LIN {X 91.990,Y -27.379,Z -185.770,A -90.000,B 90.000,C 0.000} C_DIS
LIN {X 91.908,Y -27.404,Z -186.279,A -90.000,B 90.000,C 0.000} C_DIS
LIN {X 91.890,Y -27.409,Z -186.423,A -90.000,B 90.000,C 0.000} C_DIS
LIN {X 91.690,Y -27.464,Z -187.831,A -90.000,B 90.000,C 0.000} C_DIS
LIN {X 91.648,Y -27.479,Z -188.136,A -90.000,B 90.000,C 0.000} C_DIS
LIN {X 91.626,Y -27.484,Z -188.383,A -90.000,B 90.000,C 0.000} C_DIS
LIN {X 91.538,Y -27.498,Z -189.497,A -90.000,B 90.000,C 0.000} C_DIS
LIN {X 91.494,Y -27.511,Z -190.085,A -90.000,B 90.000,C 0.000} C_DIS
LIN {X 91.464,Y -27.521,Z -190.421,A -90.000,B 90.000,C 0.000} C_DIS
LIN {X 91.445,Y -27.529,Z -190.604,A -90.000,B 90.000,C 0.000} C_DIS
LIN {X 91.394,Y -27.540,Z -191.043,A -90.000,B 90.000,C 0.000} C_DIS
LIN {X 91.332,Y -27.547,Z -191.830,A -90.000,B 90.000,C 0.000} C_DIS
LIN {X 91.227,Y -27.567,Z -193.196,A -90.000,B 90.000,C 0.000} C_DIS
LIN {X 91.184,Y -27.565,Z -193.656,A -90.000,B 90.000,C 0.000} C_DIS
LIN {X 90.969,Y -27.575,Z -195.817,A -90.000,B 90.000,C 0.000} C_DIS
LIN {X 90.925,Y -27.569,Z -196.389,A -90.000,B 90.000,C 0.000} C_DIS
LIN {X 90.877,Y -27.563,Z -196.833,A -90.000,B 90.000,C 0.000} C_DIS
LIN {X 90.590,Y -27.556,Z -198.905,A -90.000,B 90.000,C 0.000} C_DIS
LIN {X 90.465,Y -27.542,Z -199.948,A -90.000,B 90.000,C 0.000} C_DIS
LIN {X 90.447,Y -27.538,Z -200.085,A -90.000,B 90.000,C 0.000} C_DIS
LIN {X 90.408,Y -27.527,Z -200.354,A -90.000,B 90.000,C 0.000} C_DIS
LIN {X 90.390,Y -27.524,Z -200.463,A -90.000,B 90.000,C 0.000} C_DIS
LIN {X 90.100,Y -27.495,Z -202.020,A -90.000,B 90.000,C 0.000} C_DIS
LIN {X 89.684,Y -27.430,Z -204.401,A -90.000,B 90.000,C 0.000} C_DIS
LIN {X 89.653,Y -27.425,Z -204.568,A -90.000,B 90.000,C 0.000} C_DIS
LIN {X 89.484,Y -27.409,Z -205.376,A -90.000,B 90.000,C 0.000} C_DIS
LIN {X 88.923,Y -27.339,Z -208.174,A -90.000,B 90.000,C 0.000} C_DIS
LIN {X 88.721,Y -27.328,Z -209.087,A -90.000,B 90.000,C 0.000} C_DIS
LIN {X 88.664,Y -27.324,Z -209.342,A -90.000,B 90.000,C 0.000} C_DIS
LIN {X 88.255,Y -27.308,Z -211.076,A -90.000,B 90.000,C 0.000} C_DIS
LIN {X 88.255,Y -60.000,Z -211.076,A -90.000,B 90.000,C 0.000} C_DIS
LIN {X -103.369,Y -60.000,Z -243.561,A -90.000,B 90.000,C 0.000} C_DIS
LIN {X -103.369,Y -27.806,Z -243.561,A -90.000,B 90.000,C 0.000} C_DIS
LIN {X -103.055,Y -27.609,Z -243.240,A -90.000,B 90.000,C 0.000} C_DIS
LIN {X -102.608,Y -27.516,Z -242.873,A -90.000,B 90.000,C 0.000} C_DIS
LIN {X -101.362,Y -27.506,Z -241.971,A -90.000,B 90.000,C 0.000} C_DIS
LIN {X -101.122,Y -27.501,Z -241.807,A -90.000,B 90.000,C 0.000} C_DIS
LIN {X -99.449,Y -27.495,Z -240.683,A -90.000,B 90.000,C 0.000} C_DIS
LIN {X -96.335,Y -27.500,Z -238.546,A -90.000,B 90.000,C 0.000} C_DIS
LIN {X -93.712,Y -27.488,Z -236.739,A -90.000,B 90.000,C 0.000} C_DIS
LIN {X -93.290,Y -27.484,Z -236.461,A -90.000,B 90.000,C 0.000} C_DIS
LIN {X -92.213,Y -27.482,Z -235.765,A -90.000,B 90.000,C 0.000} C_DIS
LIN {X -90.517,Y -27.487,Z -234.652,A -90.000,B 90.000,C 0.000} C_DIS
LIN {X -85.124,Y -27.476,Z -231.104,A -90.000,B 90.000,C 0.000} C_DIS
LIN {X -84.873,Y -27.473,Z -230.946,A -90.000,B 90.000,C 0.000} C_DIS
LIN {X -84.774,Y -27.475,Z -230.885,A -90.000,B 90.000,C 0.000} C_DIS
LIN {X -84.558,Y -27.474,Z -230.749,A -90.000,B 90.000,C 0.000} C_DIS
LIN {X -82.273,Y -27.472,Z -229.327,A -90.000,B 90.000,C 0.000} C_DIS
LIN {X -78.940,Y -27.469,Z -227.252,A -90.000,B 90.000,C 0.000} C_DIS
LIN {X -76.872,Y -27.469,Z -225.965,A -90.000,B 90.000,C 0.000} C_DIS
LIN {X -76.380,Y -27.464,Z -225.673,A -90.000,B 90.000,C 0.000} C_DIS
LIN {X -70.507,Y -27.476,Z -222.219,A -90.000,B 90.000,C 0.000} C_DIS
LIN {X -68.311,Y -27.485,Z -220.933,A -90.000,B 90.000,C 0.000} C_DIS
LIN {X -67.723,Y -27.484,Z -220.599,A -90.000,B 90.000,C 0.000} C_DIS
LIN {X -61.693,Y -27.522,Z -217.200,A -90.000,B 90.000,C 0.000} C_DIS
LIN {X -59.270,Y -27.530,Z -215.854,A -90.000,B 90.000,C 0.000} C_DIS
LIN {X -55.292,Y -27.561,Z -213.671,A -90.000,B 90.000,C 0.000} C_DIS
LIN {X -53.229,Y -27.571,Z -212.555,A -90.000,B 90.000,C 0.000} C_DIS
LIN {X -51.847,Y -27.581,Z -211.815,A -90.000,B 90.000,C 0.000} C_DIS
LIN {X -47.655,Y -27.617,Z -209.542,A -90.000,B 90.000,C 0.000} C_DIS
LIN {X -44.795,Y -27.636,Z -208.026,A -90.000,B 90.000,C 0.000} C_DIS
LIN {X -44.368,Y -27.643,Z -207.794,A -90.000,B 90.000,C 0.000} C_DIS
LIN {X -42.572,Y -27.654,Z -206.808,A -90.000,B 90.000,C 0.000} C_DIS
LIN {X -38.988,Y -27.667,Z -204.858,A -90.000,B 90.000,C 0.000} C_DIS
LIN {X -38.628,Y -27.672,Z -204.656,A -90.000,B 90.000,C 0.000} C_DIS
LIN {X -38.069,Y -27.674,Z -204.339,A -90.000,B 90.000,C 0.000} C_DIS
LIN {X -34.183,Y -27.676,Z -202.130,A -90.000,B 90.000,C 0.000} C_DIS
LIN {X -33.519,Y -27.677,Z -201.729,A -90.000,B 90.000,C 0.000} C_DIS
LIN {X -30.256,Y -27.674,Z -199.760,A -90.000,B 90.000,C 0.000} C_DIS
LIN {X -30.194,Y -27.675,Z -199.720,A -90.000,B 90.000,C 0.000} C_DIS
LIN {X -26.908,Y -27.672,Z -197.578,A -90.000,B 90.000,C 0.000} C_DIS
LIN {X -26.646,Y -27.678,Z -197.398,A -90.000,B 90.000,C 0.000} C_DIS
LIN {X -23.666,Y -27.685,Z -195.296,A -90.000,B 90.000,C 0.000} C_DIS
LIN {X -21.311,Y -27.698,Z -193.492,A -90.000,B 90.000,C 0.000} C_DIS
LIN {X -20.756,Y -27.705,Z -193.061,A -90.000,B 90.000,C 0.000} C_DIS
LIN {X -20.525,Y -27.712,Z -192.874,A -90.000,B 90.000,C 0.000} C_DIS
LIN {X -18.379,Y -27.730,Z -191.093,A -90.000,B 90.000,C 0.000} C_DIS
LIN {X -17.666,Y -27.744,Z -190.489,A -90.000,B 90.000,C 0.000} C_DIS
LIN {X -17.400,Y -27.752,Z -190.258,A -90.000,B 90.000,C 0.000} C_DIS
LIN {X -16.396,Y -27.763,Z -189.364,A -90.000,B 90.000,C 0.000} C_DIS
LIN {X -14.874,Y -27.801,Z -187.976,A -90.000,B 90.000,C 0.000} C_DIS
LIN {X -14.452,Y -27.820,Z -187.579,A -90.000,B 90.000,C 0.000} C_DIS
LIN {X -13.143,Y -27.847,Z -186.306,A -90.000,B 90.000,C 0.000} C_DIS
LIN {X -12.383,Y -27.868,Z -185.574,A -90.000,B 90.000,C 0.000} C_DIS
LIN {X -11.697,Y -27.877,Z -184.927,A -90.000,B 90.000,C 0.000} C_DIS
LIN {X -11.309,Y -27.902,Z -184.535,A -90.000,B 90.000,C 0.000} C_DIS
LIN {X -10.955,Y -27.912,Z -184.159,A -90.000,B 90.000,C 0.000} C_DIS
LIN {X -9.538,Y -27.938,Z -182.672,A -90.000,B 90.000,C 0.000} C_DIS
LIN {X -8.754,Y -27.965,Z -181.869,A -90.000,B 90.000,C 0.000} C_DIS
LIN {X -8.149,Y -28.018,Z -181.211,A -90.000,B 90.000,C 0.000} C_DIS
LIN {X -7.812,Y -28.032,Z -180.819,A -90.000,B 90.000,C 0.000} C_DIS
LIN {X -6.414,Y -28.070,Z -179.206,A -90.000,B 90.000,C 0.000} C_DIS
LIN {X -5.991,Y -28.079,Z -178.722,A -90.000,B 90.000,C 0.000} C_DIS
LIN {X -5.438,Y -28.128,Z -178.046,A -90.000,B 90.000,C 0.000} C_DIS
LIN {X -4.765,Y -28.145,Z -177.126,A -90.000,B 90.000,C 0.000} C_DIS
LIN {X -4.342,Y -28.159,Z -176.556,A -90.000,B 90.000,C 0.000} C_DIS
LIN {X -3.482,Y -28.183,Z -175.403,A -90.000,B 90.000,C 0.000} C_DIS
LIN {X -3.179,Y -28.213,Z -174.973,A -90.000,B 90.000,C 0.000} C_DIS
LIN {X -3.054,Y -28.227,Z -174.800,A -90.000,B 90.000,C 0.000} C_DIS
LIN {X -2.768,Y -28.228,Z -174.322,A -90.000,B 90.000,C 0.000} C_DIS
LIN {X -2.310,Y -28.239,Z -173.581,A -90.000,B 90.000,C 0.000} C_DIS
LIN {X -1.574,Y -28.291,Z -172.351,A -90.000,B 90.000,C 0.000} C_DIS
LIN {X -1.394,Y -28.295,Z -172.018,A -90.000,B 90.000,C 0.000} C_DIS
LIN {X -1.247,Y -28.308,Z -171.735,A -90.000,B 90.000,C 0.000} C_DIS
LIN {X -1.150,Y -28.311,Z -171.523,A -90.000,B 90.000,C 0.000} C_DIS
LIN {X -1.055,Y -28.319,Z -171.309,A -90.000,B 90.000,C 0.000} C_DIS
LIN {X -0.727,Y -28.324,Z -170.427,A -90.000,B 90.000,C 0.000} C_DIS
LIN {X -0.556,Y -28.330,Z -169.998,A -90.000,B 90.000,C 0.000} C_DIS
LIN {X -0.131,Y -28.333,Z -168.956,A -90.000,B 90.000,C 0.000} C_DIS
LIN {X 0.016,Y -28.344,Z -168.581,A -90.000,B 90.000,C 0.000} C_DIS
LIN {X 0.075,Y -28.358,Z -168.416,A -90.000,B 90.000,C 0.000} C_DIS
LIN {X 0.321,Y -28.370,Z -167.381,A -90.000,B 90.000,C 0.000} C_DIS
LIN {X 0.403,Y -28.356,Z -166.895,A -90.000,B 90.000,C 0.000} C_DIS
LIN {X 0.614,Y -28.360,Z -165.525,A -90.000,B 90.000,C 0.000} C_DIS
LIN {X 0.613,Y -28.356,Z -165.483,A -90.000,B 90.000,C 0.000} C_DIS
LIN {X 0.543,Y -28.369,Z -164.645,A -90.000,B 90.000,C 0.000} C_DIS
LIN {X 0.477,Y -28.381,Z -163.838,A -90.000,B 90.000,C 0.000} C_DIS
LIN {X 0.445,Y -28.379,Z -163.571,A -90.000,B 90.000,C 0.000} C_DIS
LIN {X 0.261,Y -28.282,Z -163.119,A -90.000,B 90.000,C 0.000} C_DIS
LIN {X 0.200,Y -28.251,Z -162.961,A -90.000,B 90.000,C 0.000} C_DIS
LIN {X -0.226,Y -28.228,Z -162.117,A -90.000,B 90.000,C 0.000} C_DIS
LIN {X -0.493,Y -28.161,Z -161.770,A -90.000,B 90.000,C 0.000} C_DIS
LIN {X -0.916,Y -28.046,Z -161.199,A -90.000,B 90.000,C 0.000} C_DIS
LIN {X -1.178,Y -28.040,Z -160.913,A -90.000,B 90.000,C 0.000} C_DIS
LIN {X -1.412,Y -28.030,Z -160.642,A -90.000,B 90.000,C 0.000} C_DIS
LIN {X -1.913,Y -27.952,Z -160.171,A -90.000,B 90.000,C 0.000} C_DIS
LIN {X -2.368,Y -27.884,Z -159.739,A -90.000,B 90.000,C 0.000} C_DIS
LIN {X -2.403,Y -27.883,Z -159.711,A -90.000,B 90.000,C 0.000} C_DIS
LIN {X -2.661,Y -27.876,Z -159.505,A -90.000,B 90.000,C 0.000} C_DIS
LIN {X -2.941,Y -27.874,Z -159.275,A -90.000,B 90.000,C 0.000} C_DIS
LIN {X -3.035,Y -27.872,Z -159.197,A -90.000,B 90.000,C 0.000} C_DIS
LIN {X -3.740,Y -27.793,Z -158.681,A -90.000,B 90.000,C 0.000} C_DIS
LIN {X -4.065,Y -27.749,Z -158.428,A -90.000,B 90.000,C 0.000} C_DIS
LIN {X -4.255,Y -27.742,Z -158.307,A -90.000,B 90.000,C 0.000} C_DIS
LIN {X -5.243,Y -27.737,Z -157.650,A -90.000,B 90.000,C 0.000} C_DIS
LIN {X -5.356,Y -27.731,Z -157.577,A -90.000,B 90.000,C 0.000} C_DIS
LIN {X -6.117,Y -27.678,Z -157.059,A -90.000,B 90.000,C 0.000} C_DIS
LIN {X -7.097,Y -27.645,Z -156.442,A -90.000,B 90.000,C 0.000} C_DIS
LIN {X -7.589,Y -27.622,Z -156.137,A -90.000,B 90.000,C 0.000} C_DIS
LIN {X -8.273,Y -27.603,Z -155.703,A -90.000,B 90.000,C 0.000} C_DIS
LIN {X -8.376,Y -27.599,Z -155.634,A -90.000,B 90.000,C 0.000} C_DIS
LIN {X -9.611,Y -27.564,Z -154.843,A -90.000,B 90.000,C 0.000} C_DIS
LIN {X -10.209,Y -27.543,Z -154.450,A -90.000,B 90.000,C 0.000} C_DIS
LIN {X -10.831,Y -27.532,Z -154.034,A -90.000,B 90.000,C 0.000} C_DIS
LIN {X -11.149,Y -27.519,Z -153.803,A -90.000,B 90.000,C 0.000} C_DIS
LIN {X -12.438,Y -27.489,Z -152.914,A -90.000,B 90.000,C 0.000} C_DIS
LIN {X -12.864,Y -27.473,Z -152.624,A -90.000,B 90.000,C 0.000} C_DIS
LIN {X -13.338,Y -27.464,Z -152.296,A -90.000,B 90.000,C 0.000} C_DIS
LIN {X -13.599,Y -27.457,Z -152.095,A -90.000,B 90.000,C 0.000} C_DIS
LIN {X -14.698,Y -27.440,Z -151.283,A -90.000,B 90.000,C 0.000} C_DIS
LIN {X -15.643,Y -27.413,Z -150.592,A -90.000,B 90.000,C 0.000} C_DIS
LIN {X -16.148,Y -27.400,Z -150.221,A -90.000,B 90.000,C 0.000} C_DIS
LIN {X -16.592,Y -27.390,Z -149.860,A -90.000,B 90.000,C 0.000} C_DIS
LIN {X -17.132,Y -27.383,Z -149.430,A -90.000,B 90.000,C 0.000} C_DIS
LIN {X -17.811,Y -27.370,Z -148.893,A -90.000,B 90.000,C 0.000} C_DIS
LIN {X -18.518,Y -27.359,Z -148.336,A -90.000,B 90.000,C 0.000} C_DIS
LIN {X -19.270,Y -27.348,Z -147.769,A -90.000,B 90.000,C 0.000} C_DIS
LIN {X -19.598,Y -27.342,Z -147.511,A -90.000,B 90.000,C 0.000} C_DIS
LIN {X -20.875,Y -27.329,Z -146.416,A -90.000,B 90.000,C 0.000} C_DIS
LIN {X -22.706,Y -27.315,Z -144.890,A -90.000,B 90.000,C 0.000} C_DIS
LIN {X -23.017,Y -27.314,Z -144.646,A -90.000,B 90.000,C 0.000} C_DIS
LIN {X -23.794,Y -27.311,Z -143.936,A -90.000,B 90.000,C 0.000} C_DIS
LIN {X -24.478,Y -27.310,Z -143.312,A -90.000,B 90.000,C 0.000} C_DIS
LIN {X -25.785,Y -27.309,Z -142.145,A -90.000,B 90.000,C 0.000} C_DIS
LIN {X -26.511,Y -27.308,Z -141.523,A -90.000,B 90.000,C 0.000} C_DIS
LIN {X -26.720,Y -27.308,Z -141.334,A -90.000,B 90.000,C 0.000} C_DIS
LIN {X -26.793,Y -27.308,Z -141.267,A -90.000,B 90.000,C 0.000} C_DIS
LIN {X -26.898,Y -29.197,Z -141.172,A -90.000,B 90.000,C 0.000} C_DIS
LIN {X -26.911,Y -29.205,Z -141.160,A -90.000,B 90.000,C 0.000} C_DIS
LIN {X -26.913,Y -29.273,Z -141.155,A -90.000,B 90.000,C 0.000} C_DIS
LIN {X -26.925,Y -29.312,Z -141.142,A -90.000,B 90.000,C 0.000} C_DIS
LIN {X -26.959,Y -29.342,Z -141.107,A -90.000,B 90.000,C 0.000} C_DIS
LIN {X -27.026,Y -27.308,Z -141.042,A -90.000,B 90.000,C 0.000} C_DIS
LIN {X -27.144,Y -27.308,Z -140.928,A -90.000,B 90.000,C 0.000} C_DIS
LIN {X -27.161,Y -29.213,Z -140.912,A -90.000,B 90.000,C 0.000} C_DIS
LIN {X -27.163,Y -29.212,Z -140.910,A -90.000,B 90.000,C 0.000} C_DIS
LIN {X -27.166,Y -29.222,Z -140.907,A -90.000,B 90.000,C 0.000} C_DIS
LIN {X -27.182,Y -27.308,Z -140.891,A -90.000,B 90.000,C 0.000} C_DIS
LIN {X -30.222,Y -27.309,Z -137.840,A -90.000,B 90.000,C 0.000} C_DIS
LIN {X -30.549,Y -27.309,Z -137.451,A -90.000,B 90.000,C 0.000} C_DIS
LIN {X -32.741,Y -27.308,Z -134.747,A -90.000,B 90.000,C 0.000} C_DIS
LIN {X -33.107,Y -27.314,Z -134.303,A -90.000,B 90.000,C 0.000} C_DIS
LIN {X -33.314,Y -27.309,Z -134.051,A -90.000,B 90.000,C 0.000} C_DIS
LIN {X -33.612,Y -27.309,Z -133.614,A -90.000,B 90.000,C 0.000} C_DIS
LIN {X -35.907,Y -27.310,Z -130.179,A -90.000,B 90.000,C 0.000} C_DIS
LIN {X -37.253,Y -27.312,Z -127.720,A -90.000,B 90.000,C 0.000} C_DIS
LIN {X -37.408,Y -27.313,Z -127.433,A -90.000,B 90.000,C 0.000} C_DIS
LIN {X -37.959,Y -27.314,Z -126.401,A -90.000,B 90.000,C 0.000} C_DIS
LIN {X -38.164,Y -27.317,Z -126.018,A -90.000,B 90.000,C 0.000} C_DIS
LIN {X -38.966,Y -27.325,Z -124.207,A -90.000,B 90.000,C 0.000} C_DIS
LIN {X -39.268,Y -27.329,Z -123.518,A -90.000,B 90.000,C 0.000} C_DIS
LIN {X -39.615,Y -27.336,Z -122.724,A -90.000,B 90.000,C 0.000} C_DIS
LIN {X -39.769,Y -27.338,Z -122.360,A -90.000,B 90.000,C 0.000} C_DIS
LIN {X -39.971,Y -27.345,Z -121.857,A -90.000,B 90.000,C 0.000} C_DIS
LIN {X -40.184,Y -27.360,Z -121.327,A -90.000,B 90.000,C 0.000} C_DIS
LIN {X -40.315,Y -27.366,Z -120.937,A -90.000,B 90.000,C 0.000} C_DIS
LIN {X -40.403,Y -27.370,Z -120.666,A -90.000,B 90.000,C 0.000} C_DIS
LIN {X -40.826,Y -27.380,Z -119.213,A -90.000,B 90.000,C 0.000} C_DIS
LIN {X -41.157,Y -27.385,Z -118.037,A -90.000,B 90.000,C 0.000} C_DIS
LIN {X -41.283,Y -27.387,Z -117.575,A -90.000,B 90.000,C 0.000} C_DIS
LIN {X -41.314,Y -27.387,Z -117.455,A -90.000,B 90.000,C 0.000} C_DIS
LIN {X -41.529,Y -27.411,Z -116.709,A -90.000,B 90.000,C 0.000} C_DIS
LIN {X -41.881,Y -27.452,Z -115.485,A -90.000,B 90.000,C 0.000} C_DIS
LIN {X -41.924,Y -27.457,Z -115.334,A -90.000,B 90.000,C 0.000} C_DIS
LIN {X -42.227,Y -27.514,Z -114.460,A -90.000,B 90.000,C 0.000} C_DIS
LIN {X -42.520,Y -27.563,Z -113.660,A -90.000,B 90.000,C 0.000} C_DIS
LIN {X -42.555,Y -27.567,Z -113.564,A -90.000,B 90.000,C 0.000} C_DIS
LIN {X -42.730,Y -27.603,Z -113.171,A -90.000,B 90.000,C 0.000} C_DIS
LIN {X -42.874,Y -27.624,Z -112.861,A -90.000,B 90.000,C 0.000} C_DIS
LIN {X -42.965,Y -27.640,Z -112.671,A -90.000,B 90.000,C 0.000} C_DIS
LIN {X -43.317,Y -27.678,Z -111.967,A -90.000,B 90.000,C 0.000} C_DIS
LIN {X -43.517,Y -27.686,Z -111.584,A -90.000,B 90.000,C 0.000} C_DIS
LIN {X -43.555,Y -27.685,Z -111.513,A -90.000,B 90.000,C 0.000} C_DIS
LIN {X -43.660,Y -27.689,Z -111.341,A -90.000,B 90.000,C 0.000} C_DIS
LIN {X -44.234,Y -27.731,Z -110.439,A -90.000,B 90.000,C 0.000} C_DIS
LIN {X -44.344,Y -27.734,Z -110.272,A -90.000,B 90.000,C 0.000} C_DIS
LIN {X -45.008,Y -27.721,Z -109.296,A -90.000,B 90.000,C 0.000} C_DIS
LIN {X -45.128,Y -27.723,Z -109.131,A -90.000,B 90.000,C 0.000} C_DIS
LIN {X -45.591,Y -27.727,Z -108.479,A -90.000,B 90.000,C 0.000} C_DIS
LIN {X -45.928,Y -27.717,Z -108.021,A -90.000,B 90.000,C 0.000} C_DIS
LIN {X -46.530,Y -27.711,Z -107.187,A -90.000,B 90.000,C 0.000} C_DIS
LIN {X -46.929,Y -27.721,Z -106.664,A -90.000,B 90.000,C 0.000} C_DIS
LIN {X -47.127,Y -27.724,Z -106.403,A -90.000,B 90.000,C 0.000} C_DIS
LIN {X -47.530,Y -27.713,Z -105.883,A -90.000,B 90.000,C 0.000} C_DIS
LIN {X -48.012,Y -27.711,Z -105.251,A -90.000,B 90.000,C 0.000} C_DIS
LIN {X -48.754,Y -27.727,Z -104.322,A -90.000,B 90.000,C 0.000} C_DIS
LIN {X -49.134,Y -27.724,Z -103.859,A -90.000,B 90.000,C 0.000} C_DIS
LIN {X -49.367,Y -27.717,Z -103.565,A -90.000,B 90.000,C 0.000} C_DIS
LIN {X -49.765,Y -27.713,Z -103.073,A -90.000,B 90.000,C 0.000} C_DIS
LIN {X -49.990,Y -27.717,Z -102.790,A -90.000,B 90.000,C 0.000} C_DIS
LIN {X -51.040,Y -27.715,Z -101.485,A -90.000,B 90.000,C 0.000} C_DIS
LIN {X -51.428,Y -27.709,Z -100.989,A -90.000,B 90.000,C 0.000} C_DIS
LIN {X -51.547,Y -27.709,Z -100.842,A -90.000,B 90.000,C 0.000} C_DIS
LIN {X -51.805,Y -27.705,Z -100.512,A -90.000,B 90.000,C 0.000} C_DIS
LIN {X -52.097,Y -27.696,Z -100.126,A -90.000,B 90.000,C 0.000} C_DIS
LIN {X -53.332,Y -27.713,Z -98.432,A -90.000,B 90.000,C 0.000} C_DIS
LIN {X -53.687,Y -27.724,Z -97.960,A -90.000,B 90.000,C 0.000} C_DIS
LIN {X -54.103,Y -27.730,Z -97.412,A -90.000,B 90.000,C 0.000} C_DIS
LIN {X -54.366,Y -27.728,Z -97.052,A -90.000,B 90.000,C 0.000} C_DIS
LIN {X -54.897,Y -27.737,Z -96.308,A -90.000,B 90.000,C 0.000} C_DIS
LIN {X -55.218,Y -27.748,Z -95.870,A -90.000,B 90.000,C 0.000} C_DIS
LIN {X -56.401,Y -27.770,Z -94.273,A -90.000,B 90.000,C 0.000} C_DIS
LIN {X -56.592,Y -27.774,Z -94.016,A -90.000,B 90.000,C 0.000} C_DIS
LIN {X -56.744,Y -27.778,Z -93.807,A -90.000,B 90.000,C 0.000} C_DIS
LIN {X -57.102,Y -27.776,Z -93.309,A -90.000,B 90.000,C 0.000} C_DIS
LIN {X -58.057,Y -27.788,Z -91.955,A -90.000,B 90.000,C 0.000} C_DIS
LIN {X -58.231,Y -27.789,Z -91.705,A -90.000,B 90.000,C 0.000} C_DIS
LIN {X -58.545,Y -27.795,Z -91.262,A -90.000,B 90.000,C 0.000} C_DIS
LIN {X -58.727,Y -27.804,Z -90.999,A -90.000,B 90.000,C 0.000} C_DIS
LIN {X -59.582,Y -27.834,Z -89.773,A -90.000,B 90.000,C 0.000} C_DIS
LIN {X -60.304,Y -27.878,Z -88.762,A -90.000,B 90.000,C 0.000} C_DIS
LIN {X -60.643,Y -27.910,Z -88.306,A -90.000,B 90.000,C 0.000} C_DIS
LIN {X -61.350,Y -27.954,Z -87.384,A -90.000,B 90.000,C 0.000} C_DIS
LIN {X -62.230,Y -27.983,Z -86.270,A -90.000,B 90.000,C 0.000} C_DIS
LIN {X -62.389,Y -27.989,Z -86.070,A -90.000,B 90.000,C 0.000} C_DIS
LIN {X -63.199,Y -27.994,Z -85.087,A -90.000,B 90.000,C 0.000} C_DIS
LIN {X -63.468,Y -28.006,Z -84.745,A -90.000,B 90.000,C 0.000} C_DIS
LIN {X -63.673,Y -28.009,Z -84.475,A -90.000,B 90.000,C 0.000} C_DIS
LIN {X -64.048,Y -28.022,Z -83.993,A -90.000,B 90.000,C 0.000} C_DIS
LIN {X -64.314,Y -28.028,Z -83.656,A -90.000,B 90.000,C 0.000} C_DIS
LIN {X -64.753,Y -28.050,Z -83.076,A -90.000,B 90.000,C 0.000} C_DIS
LIN {X -65.187,Y -28.091,Z -82.526,A -90.000,B 90.000,C 0.000} C_DIS
LIN {X -65.475,Y -28.102,Z -82.184,A -90.000,B 90.000,C 0.000} C_DIS
LIN {X -65.758,Y -28.107,Z -81.835,A -90.000,B 90.000,C 0.000} C_DIS
LIN {X -66.105,Y -28.140,Z -81.404,A -90.000,B 90.000,C 0.000} C_DIS
LIN {X -66.407,Y -28.152,Z -81.054,A -90.000,B 90.000,C 0.000} C_DIS
LIN {X -66.771,Y -28.154,Z -80.615,A -90.000,B 90.000,C 0.000} C_DIS
LIN {X -66.835,Y -28.156,Z -80.536,A -90.000,B 90.000,C 0.000} C_DIS
LIN {X -67.132,Y -28.174,Z -80.149,A -90.000,B 90.000,C 0.000} C_DIS
LIN {X -67.591,Y -28.189,Z -79.534,A -90.000,B 90.000,C 0.000} C_DIS
LIN {X -68.739,Y -28.255,Z -77.923,A -90.000,B 90.000,C 0.000} C_DIS
LIN {X -69.084,Y -28.284,Z -77.448,A -90.000,B 90.000,C 0.000} C_DIS
LIN {X -69.329,Y -28.293,Z -77.097,A -90.000,B 90.000,C 0.000} C_DIS
LIN {X -69.702,Y -28.316,Z -76.537,A -90.000,B 90.000,C 0.000} C_DIS
LIN {X -70.129,Y -28.342,Z -75.896,A -90.000,B 90.000,C 0.000} C_DIS
LIN {X -70.383,Y -28.368,Z -75.526,A -90.000,B 90.000,C 0.000} C_DIS
LIN {X -70.764,Y -28.402,Z -74.982,A -90.000,B 90.000,C 0.000} C_DIS
LIN {X -70.884,Y -28.406,Z -74.826,A -90.000,B 90.000,C 0.000} C_DIS
LIN {X -71.247,Y -28.411,Z -74.352,A -90.000,B 90.000,C 0.000} C_DIS
LIN {X -71.617,Y -28.407,Z -73.893,A -90.000,B 90.000,C 0.000} C_DIS
LIN {X -72.102,Y -28.432,Z -73.303,A -90.000,B 90.000,C 0.000} C_DIS
LIN {X -72.834,Y -28.422,Z -72.569,A -90.000,B 90.000,C 0.000} C_DIS
LIN {X -72.966,Y -28.425,Z -72.440,A -90.000,B 90.000,C 0.000} C_DIS
LIN {X -73.130,Y -28.437,Z -72.285,A -90.000,B 90.000,C 0.000} C_DIS
LIN {X -73.444,Y -28.447,Z -71.980,A -90.000,B 90.000,C 0.000} C_DIS
LIN {X -73.601,Y -28.446,Z -71.842,A -90.000,B 90.000,C 0.000} C_DIS
LIN {X -73.772,Y -28.453,Z -71.699,A -90.000,B 90.000,C 0.000} C_DIS
LIN {X -74.003,Y -28.457,Z -71.532,A -90.000,B 90.000,C 0.000} C_DIS
LIN {X -74.407,Y -28.471,Z -71.245,A -90.000,B 90.000,C 0.000} C_DIS
LIN {X -74.532,Y -28.471,Z -71.163,A -90.000,B 90.000,C 0.000} C_DIS
LIN {X -74.824,Y -28.493,Z -70.984,A -90.000,B 90.000,C 0.000} C_DIS
LIN {X -74.932,Y -28.512,Z -70.923,A -90.000,B 90.000,C 0.000} C_DIS
LIN {X -75.008,Y -28.495,Z -70.941,A -90.000,B 90.000,C 0.000} C_DIS
LIN {X -75.159,Y -28.470,Z -70.990,A -90.000,B 90.000,C 0.000} C_DIS
LIN {X -75.302,Y -28.447,Z -71.035,A -90.000,B 90.000,C 0.000} C_DIS
LIN {X -75.419,Y -28.436,Z -71.075,A -90.000,B 90.000,C 0.000} C_DIS
LIN {X -75.526,Y -28.428,Z -71.108,A -90.000,B 90.000,C 0.000} C_DIS
LIN {X -75.715,Y -28.415,Z -71.162,A -90.000,B 90.000,C 0.000} C_DIS
LIN {X -75.995,Y -28.393,Z -71.241,A -90.000,B 90.000,C 0.000} C_DIS
LIN {X -76.053,Y -28.389,Z -71.257,A -90.000,B 90.000,C 0.000} C_DIS
LIN {X -76.236,Y -28.380,Z -71.302,A -90.000,B 90.000,C 0.000} C_DIS
LIN {X -76.473,Y -28.369,Z -71.353,A -90.000,B 90.000,C 0.000} C_DIS
LIN {X -76.715,Y -28.361,Z -71.401,A -90.000,B 90.000,C 0.000} C_DIS
LIN {X -76.847,Y -28.352,Z -71.423,A -90.000,B 90.000,C 0.000} C_DIS
LIN {X -77.146,Y -28.335,Z -71.464,A -90.000,B 90.000,C 0.000} C_DIS
LIN {X -77.393,Y -28.322,Z -71.492,A -90.000,B 90.000,C 0.000} C_DIS
LIN {X -77.537,Y -28.318,Z -71.503,A -90.000,B 90.000,C 0.000} C_DIS
LIN {X -77.870,Y -28.296,Z -71.509,A -90.000,B 90.000,C 0.000} C_DIS
LIN {X -78.006,Y -28.289,Z -71.508,A -90.000,B 90.000,C 0.000} C_DIS
LIN {X -78.336,Y -28.279,Z -71.494,A -90.000,B 90.000,C 0.000} C_DIS
LIN {X -78.470,Y -28.270,Z -71.486,A -90.000,B 90.000,C 0.000} C_DIS
LIN {X -78.586,Y -28.264,Z -71.475,A -90.000,B 90.000,C 0.000} C_DIS
LIN {X -78.727,Y -28.259,Z -71.459,A -90.000,B 90.000,C 0.000} C_DIS
LIN {X -78.995,Y -28.245,Z -71.425,A -90.000,B 90.000,C 0.000} C_DIS
LIN {X -79.034,Y -28.243,Z -71.418,A -90.000,B 90.000,C 0.000} C_DIS
LIN {X -79.208,Y -28.237,Z -71.379,A -90.000,B 90.000,C 0.000} C_DIS
LIN {X -79.548,Y -28.226,Z -71.290,A -90.000,B 90.000,C 0.000} C_DIS
LIN {X -79.782,Y -28.224,Z -71.219,A -90.000,B 90.000,C 0.000} C_DIS
LIN {X -80.088,Y -28.204,Z -71.111,A -90.000,B 90.000,C 0.000} C_DIS
LIN {X -80.152,Y -28.201,Z -71.086,A -90.000,B 90.000,C 0.000} C_DIS
LIN {X -80.472,Y -28.180,Z -70.944,A -90.000,B 90.000,C 0.000} C_DIS
LIN {X -80.555,Y -28.176,Z -70.906,A -90.000,B 90.000,C 0.000} C_DIS
LIN {X -80.623,Y -28.174,Z -70.871,A -90.000,B 90.000,C 0.000} C_DIS
LIN {X -80.984,Y -28.164,Z -70.660,A -90.000,B 90.000,C 0.000} C_DIS
LIN {X -81.049,Y -28.163,Z -70.620,A -90.000,B 90.000,C 0.000} C_DIS
LIN {X -81.148,Y -28.157,Z -70.548,A -90.000,B 90.000,C 0.000} C_DIS
LIN {X -81.374,Y -28.149,Z -70.372,A -90.000,B 90.000,C 0.000} C_DIS
LIN {X -81.573,Y -28.128,Z -70.203,A -90.000,B 90.000,C 0.000} C_DIS
LIN {X -81.818,Y -28.105,Z -69.993,A -90.000,B 90.000,C 0.000} C_DIS
LIN {X -81.935,Y -28.097,Z -69.884,A -90.000,B 90.000,C 0.000} C_DIS
LIN {X -82.044,Y -28.094,Z -69.772,A -90.000,B 90.000,C 0.000} C_DIS
LIN {X -82.209,Y -28.077,Z -69.584,A -90.000,B 90.000,C 0.000} C_DIS
LIN {X -82.296,Y -28.069,Z -69.478,A -90.000,B 90.000,C 0.000} C_DIS
LIN {X -82.410,Y -28.050,Z -69.324,A -90.000,B 90.000,C 0.000} C_DIS
LIN {X -82.465,Y -28.043,Z -69.244,A -90.000,B 90.000,C 0.000} C_DIS
LIN {X -82.520,Y -28.036,Z -69.157,A -90.000,B 90.000,C 0.000} C_DIS
LIN {X -82.613,Y -28.030,Z -69.018,A -90.000,B 90.000,C 0.000} C_DIS
LIN {X -82.709,Y -28.022,Z -68.869,A -90.000,B 90.000,C 0.000} C_DIS
LIN {X -82.798,Y -28.016,Z -68.725,A -90.000,B 90.000,C 0.000} C_DIS
LIN {X -82.988,Y -27.977,Z -68.373,A -90.000,B 90.000,C 0.000} C_DIS
LIN {X -83.037,Y -27.961,Z -68.259,A -90.000,B 90.000,C 0.000} C_DIS
LIN {X -83.075,Y -27.957,Z -68.179,A -90.000,B 90.000,C 0.000} C_DIS
LIN {X -83.198,Y -27.947,Z -67.925,A -90.000,B 90.000,C 0.000} C_DIS
LIN {X -83.316,Y -27.933,Z -67.655,A -90.000,B 90.000,C 0.000} C_DIS
LIN {X -83.352,Y -27.931,Z -67.558,A -90.000,B 90.000,C 0.000} C_DIS
LIN {X -83.386,Y -27.930,Z -67.462,A -90.000,B 90.000,C 0.000} C_DIS
LIN {X -83.512,Y -27.924,Z -67.098,A -90.000,B 90.000,C 0.000} C_DIS
LIN {X -83.556,Y -27.918,Z -66.959,A -90.000,B 90.000,C 0.000} C_DIS
LIN {X -83.664,Y -27.913,Z -66.592,A -90.000,B 90.000,C 0.000} C_DIS
LIN {X -83.711,Y -27.904,Z -66.432,A -90.000,B 90.000,C 0.000} C_DIS
LIN {X -83.792,Y -27.881,Z -66.144,A -90.000,B 90.000,C 0.000} C_DIS
LIN {X -83.830,Y -27.873,Z -65.990,A -90.000,B 90.000,C 0.000} C_DIS
LIN {X -83.856,Y -27.863,Z -65.890,A -90.000,B 90.000,C 0.000} C_DIS
LIN {X -83.889,Y -27.849,Z -65.780,A -90.000,B 90.000,C 0.000} C_DIS
LIN {X -83.944,Y -27.814,Z -65.561,A -90.000,B 90.000,C 0.000} C_DIS
LIN {X -83.966,Y -27.801,Z -65.472,A -90.000,B 90.000,C 0.000} C_DIS
LIN {X -83.998,Y -27.788,Z -65.355,A -90.000,B 90.000,C 0.000} C_DIS
LIN {X -84.049,Y -27.775,Z -65.194,A -90.000,B 90.000,C 0.000} C_DIS
LIN {X -84.211,Y -27.768,Z -64.768,A -90.000,B 90.000,C 0.000} C_DIS
LIN {X -84.244,Y -27.768,Z -64.677,A -90.000,B 90.000,C 0.000} C_DIS
LIN {X -84.429,Y -27.771,Z -64.103,A -90.000,B 90.000,C 0.000} C_DIS
LIN {X -84.485,Y -27.775,Z -63.916,A -90.000,B 90.000,C 0.000} C_DIS
LIN {X -84.560,Y -27.779,Z -63.598,A -90.000,B 90.000,C 0.000} C_DIS
LIN {X -84.657,Y -27.793,Z -63.150,A -90.000,B 90.000,C 0.000} C_DIS
LIN {X -84.727,Y -27.818,Z -62.841,A -90.000,B 90.000,C 0.000} C_DIS
LIN {X -84.783,Y -27.843,Z -62.612,A -90.000,B 90.000,C 0.000} C_DIS
LIN {X -84.815,Y -27.861,Z -62.500,A -90.000,B 90.000,C 0.000} C_DIS
LIN {X -84.854,Y -27.886,Z -62.400,A -90.000,B 90.000,C 0.000} C_DIS
LIN {X -84.896,Y -27.910,Z -62.286,A -90.000,B 90.000,C 0.000} C_DIS
LIN {X -84.934,Y -27.930,Z -62.185,A -90.000,B 90.000,C 0.000} C_DIS
LIN {X -84.991,Y -27.964,Z -62.055,A -90.000,B 90.000,C 0.000} C_DIS
LIN {X -85.046,Y -28.003,Z -61.915,A -90.000,B 90.000,C 0.000} C_DIS
LIN {X -85.120,Y -28.066,Z -61.710,A -90.000,B 90.000,C 0.000} C_DIS
LIN {X -85.152,Y -28.088,Z -61.629,A -90.000,B 90.000,C 0.000} C_DIS
LIN {X -85.167,Y -28.098,Z -61.591,A -90.000,B 90.000,C 0.000} C_DIS
LIN {X -85.193,Y -28.109,Z -61.538,A -90.000,B 90.000,C 0.000} C_DIS
LIN {X -85.237,Y -28.130,Z -61.454,A -90.000,B 90.000,C 0.000} C_DIS
LIN {X -85.349,Y -28.181,Z -61.228,A -90.000,B 90.000,C 0.000} C_DIS
LIN {X -85.597,Y -28.249,Z -60.809,A -90.000,B 90.000,C 0.000} C_DIS
LIN {X -85.726,Y -28.294,Z -60.573,A -90.000,B 90.000,C 0.000} C_DIS
LIN {X -85.738,Y -28.298,Z -60.549,A -90.000,B 90.000,C 0.000} C_DIS
LIN {X -85.893,Y -28.321,Z -60.298,A -90.000,B 90.000,C 0.000} C_DIS
LIN {X -85.935,Y -28.329,Z -60.229,A -90.000,B 90.000,C 0.000} C_DIS
LIN {X -86.415,Y -28.448,Z -59.455,A -90.000,B 90.000,C 0.000} C_DIS
LIN {X -86.480,Y -28.461,Z -59.356,A -90.000,B 90.000,C 0.000} C_DIS
LIN {X -86.677,Y -28.497,Z -59.047,A -90.000,B 90.000,C 0.000} C_DIS
LIN {X -86.830,Y -28.518,Z -58.799,A -90.000,B 90.000,C 0.000} C_DIS
LIN {X -87.003,Y -28.549,Z -58.501,A -90.000,B 90.000,C 0.000} C_DIS
LIN {X -87.219,Y -28.598,Z -58.108,A -90.000,B 90.000,C 0.000} C_DIS
LIN {X -87.414,Y -28.635,Z -57.743,A -90.000,B 90.000,C 0.000} C_DIS
LIN {X -87.492,Y -28.651,Z -57.585,A -90.000,B 90.000,C 0.000} C_DIS
LIN {X -87.742,Y -28.696,Z -57.058,A -90.000,B 90.000,C 0.000} C_DIS
LIN {X -87.785,Y -28.705,Z -56.963,A -90.000,B 90.000,C 0.000} C_DIS
LIN {X -87.825,Y -28.715,Z -56.867,A -90.000,B 90.000,C 0.000} C_DIS
LIN {X -87.907,Y -28.738,Z -56.655,A -90.000,B 90.000,C 0.000} C_DIS
LIN {X -87.939,Y -28.747,Z -56.565,A -90.000,B 90.000,C 0.000} C_DIS
LIN {X -88.058,Y -28.781,Z -56.170,A -90.000,B 90.000,C 0.000} C_DIS
LIN {X -88.132,Y -28.797,Z -55.919,A -90.000,B 90.000,C 0.000} C_DIS
LIN {X -88.161,Y -28.807,Z -55.791,A -90.000,B 90.000,C 0.000} C_DIS
LIN {X -88.187,Y -28.822,Z -55.631,A -90.000,B 90.000,C 0.000} C_DIS
LIN {X -88.212,Y -28.836,Z -55.463,A -90.000,B 90.000,C 0.000} C_DIS
LIN {X -88.229,Y -28.852,Z -55.293,A -90.000,B 90.000,C 0.000} C_DIS
LIN {X -88.232,Y -28.860,Z -55.214,A -90.000,B 90.000,C 0.000} C_DIS
LIN {X -88.263,Y -28.878,Z -54.962,A -90.000,B 90.000,C 0.000} C_DIS
LIN {X -88.272,Y -28.884,Z -54.877,A -90.000,B 90.000,C 0.000} C_DIS
LIN {X -88.275,Y -28.885,Z -54.819,A -90.000,B 90.000,C 0.000} C_DIS
LIN {X -88.277,Y -28.893,Z -54.698,A -90.000,B 90.000,C 0.000} C_DIS
LIN {X -88.267,Y -28.913,Z -54.445,A -90.000,B 90.000,C 0.000} C_DIS
LIN {X -88.257,Y -28.922,Z -54.237,A -90.000,B 90.000,C 0.000} C_DIS
LIN {X -88.254,Y -28.921,Z -54.189,A -90.000,B 90.000,C 0.000} C_DIS
LIN {X -88.216,Y -28.939,Z -53.830,A -90.000,B 90.000,C 0.000} C_DIS
LIN {X -88.188,Y -28.941,Z -53.676,A -90.000,B 90.000,C 0.000} C_DIS
LIN {X -88.150,Y -28.944,Z -53.501,A -90.000,B 90.000,C 0.000} C_DIS
LIN {X -88.131,Y -28.946,Z -53.422,A -90.000,B 90.000,C 0.000} C_DIS
LIN {X -88.103,Y -28.949,Z -53.324,A -90.000,B 90.000,C 0.000} C_DIS
LIN {X -88.072,Y -28.954,Z -53.233,A -90.000,B 90.000,C 0.000} C_DIS
LIN {X -88.024,Y -28.956,Z -53.117,A -90.000,B 90.000,C 0.000} C_DIS
LIN {X -87.962,Y -28.959,Z -52.978,A -90.000,B 90.000,C 0.000} C_DIS
LIN {X -87.899,Y -28.961,Z -52.851,A -90.000,B 90.000,C 0.000} C_DIS
LIN {X -87.799,Y -28.965,Z -52.665,A -90.000,B 90.000,C 0.000} C_DIS
LIN {X -87.743,Y -28.965,Z -52.573,A -90.000,B 90.000,C 0.000} C_DIS
LIN {X -87.686,Y -28.967,Z -52.488,A -90.000,B 90.000,C 0.000} C_DIS
LIN {X -87.592,Y -28.965,Z -52.367,A -90.000,B 90.000,C 0.000} C_DIS
LIN {X -87.542,Y -28.965,Z -52.310,A -90.000,B 90.000,C 0.000} C_DIS
LIN {X -87.362,Y -28.956,Z -52.126,A -90.000,B 90.000,C 0.000} C_DIS
LIN {X -87.343,Y -28.955,Z -52.107,A -90.000,B 90.000,C 0.000} C_DIS
LIN {X -87.206,Y -28.943,Z -51.986,A -90.000,B 90.000,C 0.000} C_DIS
LIN {X -87.175,Y -28.940,Z -51.962,A -90.000,B 90.000,C 0.000} C_DIS
LIN {X -87.080,Y -28.933,Z -51.893,A -90.000,B 90.000,C 0.000} C_DIS
LIN {X -86.958,Y -28.925,Z -51.816,A -90.000,B 90.000,C 0.000} C_DIS
LIN {X -86.878,Y -28.921,Z -51.772,A -90.000,B 90.000,C 0.000} C_DIS
LIN {X -86.713,Y -28.908,Z -51.682,A -90.000,B 90.000,C 0.000} C_DIS
LIN {X -86.459,Y -28.870,Z -51.550,A -90.000,B 90.000,C 0.000} C_DIS
LIN {X -86.251,Y -28.839,Z -51.449,A -90.000,B 90.000,C 0.000} C_DIS
LIN {X -86.129,Y -28.819,Z -51.396,A -90.000,B 90.000,C 0.000} C_DIS
LIN {X -85.932,Y -28.775,Z -51.318,A -90.000,B 90.000,C 0.000} C_DIS
LIN {X -85.814,Y -28.750,Z -51.279,A -90.000,B 90.000,C 0.000} C_DIS
LIN {X -85.742,Y -28.736,Z -51.258,A -90.000,B 90.000,C 0.000} C_DIS
LIN {X -85.667,Y -28.722,Z -51.238,A -90.000,B 90.000,C 0.000} C_DIS
LIN {X -85.555,Y -28.705,Z -51.216,A -90.000,B 90.000,C 0.000} C_DIS
LIN {X -85.289,Y -28.665,Z -51.169,A -90.000,B 90.000,C 0.000} C_DIS
LIN {X -85.138,Y -28.646,Z -51.151,A -90.000,B 90.000,C 0.000} C_DIS
LIN {X -85.025,Y -28.630,Z -51.146,A -90.000,B 90.000,C 0.000} C_DIS
LIN {X -84.912,Y -28.617,Z -51.147,A -90.000,B 90.000,C 0.000} C_DIS
LIN {X -84.696,Y -28.588,Z -51.156,A -90.000,B 90.000,C 0.000} C_DIS
LIN {X -84.574,Y -28.573,Z -51.163,A -90.000,B 90.000,C 0.000} C_DIS
LIN {X -84.351,Y -28.552,Z -51.188,A -90.000,B 90.000,C 0.000} C_DIS
LIN {X -84.193,Y -28.542,Z -51.217,A -90.000,B 90.000,C 0.000} C_DIS
LIN {X -83.608,Y -28.478,Z -51.335,A -90.000,B 90.000,C 0.000} C_DIS
LIN {X -83.509,Y -28.462,Z -51.358,A -90.000,B 90.000,C 0.000} C_DIS
LIN {X -83.398,Y -28.447,Z -51.387,A -90.000,B 90.000,C 0.000} C_DIS
LIN {X -83.045,Y -28.408,Z -51.494,A -90.000,B 90.000,C 0.000} C_DIS
LIN {X -82.395,Y -28.343,Z -51.708,A -90.000,B 90.000,C 0.000} C_DIS
LIN {X -82.098,Y -28.314,Z -51.810,A -90.000,B 90.000,C 0.000} C_DIS
LIN {X -81.758,Y -28.284,Z -51.933,A -90.000,B 90.000,C 0.000} C_DIS
LIN {X -81.598,Y -28.271,Z -51.999,A -90.000,B 90.000,C 0.000} C_DIS
LIN {X -81.386,Y -28.261,Z -52.097,A -90.000,B 90.000,C 0.000} C_DIS
LIN {X -81.274,Y -28.257,Z -52.150,A -90.000,B 90.000,C 0.000} C_DIS
LIN {X -81.125,Y -28.249,Z -52.224,A -90.000,B 90.000,C 0.000} C_DIS
LIN {X -80.315,Y -28.188,Z -52.643,A -90.000,B 90.000,C 0.000} C_DIS
LIN {X -80.209,Y -28.182,Z -52.701,A -90.000,B 90.000,C 0.000} C_DIS
LIN {X -79.527,Y -28.142,Z -53.108,A -90.000,B 90.000,C 0.000} C_DIS
LIN {X -79.328,Y -28.137,Z -53.224,A -90.000,B 90.000,C 0.000} C_DIS
LIN {X -79.192,Y -28.137,Z -53.308,A -90.000,B 90.000,C 0.000} C_DIS
LIN {X -79.098,Y -28.133,Z -53.372,A -90.000,B 90.000,C 0.000} C_DIS
LIN {X -78.705,Y -28.123,Z -53.655,A -90.000,B 90.000,C 0.000} C_DIS
LIN {X -77.731,Y -28.139,Z -54.320,A -90.000,B 90.000,C 0.000} C_DIS
LIN {X -77.618,Y -28.142,Z -54.403,A -90.000,B 90.000,C 0.000} C_DIS
LIN {X -77.558,Y -28.146,Z -54.443,A -90.000,B 90.000,C 0.000} C_DIS
LIN {X -77.404,Y -28.152,Z -54.554,A -90.000,B 90.000,C 0.000} C_DIS
LIN {X -77.310,Y -28.160,Z -54.626,A -90.000,B 90.000,C 0.000} C_DIS
LIN {X -77.269,Y -28.165,Z -54.656,A -90.000,B 90.000,C 0.000} C_DIS
LIN {X -77.065,Y -28.182,Z -54.797,A -90.000,B 90.000,C 0.000} C_DIS
LIN {X -76.848,Y -28.198,Z -54.947,A -90.000,B 90.000,C 0.000} C_DIS
LIN {X -76.301,Y -28.282,Z -55.297,A -90.000,B 90.000,C 0.000} C_DIS
LIN {X -76.039,Y -28.337,Z -55.459,A -90.000,B 90.000,C 0.000} C_DIS
LIN {X -75.742,Y -28.406,Z -55.659,A -90.000,B 90.000,C 0.000} C_DIS
LIN {X -75.708,Y -28.414,Z -55.683,A -90.000,B 90.000,C 0.000} C_DIS
LIN {X -75.636,Y -28.424,Z -55.722,A -90.000,B 90.000,C 0.000} C_DIS
LIN {X -75.404,Y -28.475,Z -55.835,A -90.000,B 90.000,C 0.000} C_DIS
LIN {X -75.295,Y -28.501,Z -55.893,A -90.000,B 90.000,C 0.000} C_DIS
LIN {X -75.030,Y -28.544,Z -55.985,A -90.000,B 90.000,C 0.000} C_DIS
LIN {X -74.613,Y -28.590,Z -56.075,A -90.000,B 90.000,C 0.000} C_DIS
LIN {X -74.515,Y -28.602,Z -56.099,A -90.000,B 90.000,C 0.000} C_DIS
LIN {X -73.614,Y -28.647,Z -56.166,A -90.000,B 90.000,C 0.000} C_DIS
LIN {X -73.450,Y -28.649,Z -56.164,A -90.000,B 90.000,C 0.000} C_DIS
LIN {X -73.388,Y -28.653,Z -56.162,A -90.000,B 90.000,C 0.000} C_DIS
LIN {X -72.451,Y -28.673,Z -56.023,A -90.000,B 90.000,C 0.000} C_DIS
LIN {X -71.902,Y -28.687,Z -55.948,A -90.000,B 90.000,C 0.000} C_DIS
LIN {X -71.464,Y -28.706,Z -55.886,A -90.000,B 90.000,C 0.000} C_DIS
LIN {X -70.994,Y -28.718,Z -55.775,A -90.000,B 90.000,C 0.000} C_DIS
LIN {X -70.818,Y -28.725,Z -55.735,A -90.000,B 90.000,C 0.000} C_DIS
LIN {X -70.006,Y -28.760,Z -55.566,A -90.000,B 90.000,C 0.000} C_DIS
LIN {X -69.667,Y -28.767,Z -55.481,A -90.000,B 90.000,C 0.000} C_DIS
LIN {X -69.178,Y -28.784,Z -55.356,A -90.000,B 90.000,C 0.000} C_DIS
LIN {X -68.335,Y -28.801,Z -55.081,A -90.000,B 90.000,C 0.000} C_DIS
LIN {X -68.042,Y -28.809,Z -54.985,A -90.000,B 90.000,C 0.000} C_DIS
LIN {X -67.797,Y -28.812,Z -54.888,A -90.000,B 90.000,C 0.000} C_DIS
LIN {X -66.711,Y -28.843,Z -54.527,A -90.000,B 90.000,C 0.000} C_DIS
LIN {X -66.137,Y -28.847,Z -54.299,A -90.000,B 90.000,C 0.000} C_DIS
LIN {X -65.589,Y -28.851,Z -54.087,A -90.000,B 90.000,C 0.000} C_DIS
LIN {X -64.723,Y -28.836,Z -53.713,A -90.000,B 90.000,C 0.000} C_DIS
LIN {X -64.536,Y -28.834,Z -53.632,A -90.000,B 90.000,C 0.000} C_DIS
LIN {X -64.408,Y -28.834,Z -53.582,A -90.000,B 90.000,C 0.000} C_DIS
LIN {X -64.109,Y -28.835,Z -53.475,A -90.000,B 90.000,C 0.000} C_DIS
LIN {X -63.089,Y -28.803,Z -53.123,A -90.000,B 90.000,C 0.000} C_DIS
LIN {X -62.732,Y -28.785,Z -53.002,A -90.000,B 90.000,C 0.000} C_DIS
LIN {X -62.575,Y -28.779,Z -52.955,A -90.000,B 90.000,C 0.000} C_DIS
LIN {X -61.979,Y -28.760,Z -52.805,A -90.000,B 90.000,C 0.000} C_DIS
LIN {X -61.293,Y -28.734,Z -52.634,A -90.000,B 90.000,C 0.000} C_DIS
LIN {X -60.914,Y -28.702,Z -52.547,A -90.000,B 90.000,C 0.000} C_DIS
LIN {X -60.694,Y -28.686,Z -52.502,A -90.000,B 90.000,C 0.000} C_DIS
LIN {X -60.571,Y -28.678,Z -52.481,A -90.000,B 90.000,C 0.000} C_DIS
LIN {X -60.250,Y -28.663,Z -52.436,A -90.000,B 90.000,C 0.000} C_DIS
LIN {X -60.160,Y -28.659,Z -52.427,A -90.000,B 90.000,C 0.000} C_DIS
LIN {X -59.981,Y -28.654,Z -52.411,A -90.000,B 90.000,C 0.000} C_DIS
LIN {X -58.631,Y -28.577,Z -52.306,A -90.000,B 90.000,C 0.000} C_DIS
LIN {X -58.527,Y -28.572,Z -52.300,A -90.000,B 90.000,C 0.000} C_DIS
LIN {X -57.728,Y -28.542,Z -52.278,A -90.000,B 90.000,C 0.000} C_DIS
LIN {X -57.521,Y -28.532,Z -52.273,A -90.000,B 90.000,C 0.000} C_DIS
LIN {X -57.313,Y -28.519,Z -52.270,A -90.000,B 90.000,C 0.000} C_DIS
LIN {X -57.203,Y -28.513,Z -52.271,A -90.000,B 90.000,C 0.000} C_DIS
LIN {X -56.222,Y -28.468,Z -52.308,A -90.000,B 90.000,C 0.000} C_DIS
LIN {X -55.860,Y -28.451,Z -52.322,A -90.000,B 90.000,C 0.000} C_DIS
LIN {X -55.451,Y -28.427,Z -52.342,A -90.000,B 90.000,C 0.000} C_DIS
LIN {X -54.736,Y -28.394,Z -52.393,A -90.000,B 90.000,C 0.000} C_DIS
LIN {X -54.167,Y -28.354,Z -52.444,A -90.000,B 90.000,C 0.000} C_DIS
LIN {X -53.590,Y -28.319,Z -52.500,A -90.000,B 90.000,C 0.000} C_DIS
LIN {X -53.364,Y -28.307,Z -52.522,A -90.000,B 90.000,C 0.000} C_DIS
LIN {X -52.988,Y -28.290,Z -52.564,A -90.000,B 90.000,C 0.000} C_DIS
LIN {X -52.199,Y -28.268,Z -52.672,A -90.000,B 90.000,C 0.000} C_DIS
LIN {X -52.035,Y -28.262,Z -52.695,A -90.000,B 90.000,C 0.000} C_DIS
LIN {X -51.007,Y -28.217,Z -52.847,A -90.000,B 90.000,C 0.000} C_DIS
LIN {X -50.477,Y -28.198,Z -52.930,A -90.000,B 90.000,C 0.000} C_DIS
LIN {X -48.888,Y -28.132,Z -53.202,A -90.000,B 90.000,C 0.000} C_DIS
LIN {X -48.117,Y -28.096,Z -53.338,A -90.000,B 90.000,C 0.000} C_DIS
LIN {X -47.846,Y -28.082,Z -53.388,A -90.000,B 90.000,C 0.000} C_DIS
LIN {X -45.794,Y -28.026,Z -53.820,A -90.000,B 90.000,C 0.000} C_DIS
LIN {X -43.734,Y -28.000,Z -54.291,A -90.000,B 90.000,C 0.000} C_DIS
LIN {X -42.934,Y -28.002,Z -54.465,A -90.000,B 90.000,C 0.000} C_DIS
LIN {X -42.624,Y -28.015,Z -54.526,A -90.000,B 90.000,C 0.000} C_DIS
LIN {X -41.532,Y -28.082,Z -54.726,A -90.000,B 90.000,C 0.000} C_DIS
LIN {X -40.017,Y -28.181,Z -55.023,A -90.000,B 90.000,C 0.000} C_DIS
LIN {X -38.826,Y -28.258,Z -55.262,A -90.000,B 90.000,C 0.000} C_DIS
LIN {X -37.119,Y -28.358,Z -55.619,A -90.000,B 90.000,C 0.000} C_DIS
LIN {X -35.954,Y -28.426,Z -55.866,A -90.000,B 90.000,C 0.000} C_DIS
LIN {X -35.452,Y -28.446,Z -55.964,A -90.000,B 90.000,C 0.000} C_DIS
LIN {X -34.984,Y -28.457,Z -56.060,A -90.000,B 90.000,C 0.000} C_DIS
LIN {X -34.338,Y -28.458,Z -56.160,A -90.000,B 90.000,C 0.000} C_DIS
LIN {X -32.550,Y -28.428,Z -56.370,A -90.000,B 90.000,C 0.000} C_DIS
LIN {X -32.221,Y -28.420,Z -56.410,A -90.000,B 90.000,C 0.000} C_DIS
LIN {X -31.357,Y -28.406,Z -56.527,A -90.000,B 90.000,C 0.000} C_DIS
LIN {X -29.765,Y -28.374,Z -56.745,A -90.000,B 90.000,C 0.000} C_DIS
LIN {X -29.304,Y -28.368,Z -56.806,A -90.000,B 90.000,C 0.000} C_DIS
LIN {X -27.956,Y -28.331,Z -56.991,A -90.000,B 90.000,C 0.000} C_DIS
LIN {X -27.294,Y -28.318,Z -57.090,A -90.000,B 90.000,C 0.000} C_DIS
LIN {X -26.984,Y -28.314,Z -57.135,A -90.000,B 90.000,C 0.000} C_DIS
LIN {X -26.449,Y -28.295,Z -57.194,A -90.000,B 90.000,C 0.000} C_DIS
LIN {X -25.621,Y -28.273,Z -57.280,A -90.000,B 90.000,C 0.000} C_DIS
LIN {X -25.236,Y -28.265,Z -57.324,A -90.000,B 90.000,C 0.000} C_DIS
LIN {X -24.972,Y -28.251,Z -57.332,A -90.000,B 90.000,C 0.000} C_DIS
LIN {X -24.224,Y -28.217,Z -57.353,A -90.000,B 90.000,C 0.000} C_DIS
LIN {X -23.994,Y -28.211,Z -57.366,A -90.000,B 90.000,C 0.000} C_DIS
LIN {X -23.764,Y -28.186,Z -57.346,A -90.000,B 90.000,C 0.000} C_DIS
LIN {X -23.288,Y -28.167,Z -57.312,A -90.000,B 90.000,C 0.000} C_DIS
LIN {X -23.201,Y -28.154,Z -57.291,A -90.000,B 90.000,C 0.000} C_DIS
LIN {X -23.024,Y -28.131,Z -57.255,A -90.000,B 90.000,C 0.000} C_DIS
LIN {X -22.761,Y -28.101,Z -57.208,A -90.000,B 90.000,C 0.000} C_DIS
LIN {X -22.660,Y -28.082,Z -57.178,A -90.000,B 90.000,C 0.000} C_DIS
LIN {X -22.511,Y -28.055,Z -57.137,A -90.000,B 90.000,C 0.000} C_DIS
LIN {X -21.989,Y -27.983,Z -56.981,A -90.000,B 90.000,C 0.000} C_DIS
LIN {X -21.866,Y -27.958,Z -56.935,A -90.000,B 90.000,C 0.000} C_DIS
LIN {X -21.552,Y -27.898,Z -56.829,A -90.000,B 90.000,C 0.000} C_DIS
LIN {X -20.719,Y -27.796,Z -56.500,A -90.000,B 90.000,C 0.000} C_DIS
LIN {X -19.578,Y -27.729,Z -55.972,A -90.000,B 90.000,C 0.000} C_DIS
LIN {X -19.475,Y -27.726,Z -55.925,A -90.000,B 90.000,C 0.000} C_DIS
LIN {X -18.578,Y -27.721,Z -55.522,A -90.000,B 90.000,C 0.000} C_DIS
LIN {X -18.200,Y -27.719,Z -55.353,A -90.000,B 90.000,C 0.000} C_DIS
LIN {X -17.679,Y -27.723,Z -55.127,A -90.000,B 90.000,C 0.000} C_DIS
LIN {X -17.392,Y -27.718,Z -55.014,A -90.000,B 90.000,C 0.000} C_DIS
LIN {X -16.997,Y -27.715,Z -54.862,A -90.000,B 90.000,C 0.000} C_DIS
LIN {X -16.894,Y -27.717,Z -54.824,A -90.000,B 90.000,C 0.000} C_DIS
LIN {X -16.426,Y -27.735,Z -54.661,A -90.000,B 90.000,C 0.000} C_DIS
LIN {X -15.525,Y -27.768,Z -54.353,A -90.000,B 90.000,C 0.000} C_DIS
LIN {X -15.101,Y -27.770,Z -54.224,A -90.000,B 90.000,C 0.000} C_DIS
LIN {X -14.797,Y -27.762,Z -54.146,A -90.000,B 90.000,C 0.000} C_DIS
LIN {X -14.304,Y -27.756,Z -54.026,A -90.000,B 90.000,C 0.000} C_DIS
LIN {X -13.861,Y -27.755,Z -53.921,A -90.000,B 90.000,C 0.000} C_DIS
LIN {X -13.754,Y -27.758,Z -53.898,A -90.000,B 90.000,C 0.000} C_DIS
LIN {X -13.477,Y -27.771,Z -53.842,A -90.000,B 90.000,C 0.000} C_DIS
LIN {X -13.399,Y -27.777,Z -53.828,A -90.000,B 90.000,C 0.000} C_DIS
LIN {X -12.682,Y -27.814,Z -53.710,A -90.000,B 90.000,C 0.000} C_DIS
LIN {X -12.344,Y -27.840,Z -53.662,A -90.000,B 90.000,C 0.000} C_DIS
LIN {X -11.970,Y -27.859,Z -53.624,A -90.000,B 90.000,C 0.000} C_DIS
LIN {X -11.530,Y -27.865,Z -53.597,A -90.000,B 90.000,C 0.000} C_DIS
LIN {X -11.016,Y -27.866,Z -53.562,A -90.000,B 90.000,C 0.000} C_DIS
LIN {X -10.481,Y -27.859,Z -53.534,A -90.000,B 90.000,C 0.000} C_DIS
LIN {X -10.291,Y -27.856,Z -53.529,A -90.000,B 90.000,C 0.000} C_DIS
LIN {X -9.701,Y -27.861,Z -53.525,A -90.000,B 90.000,C 0.000} C_DIS
LIN {X -9.503,Y -27.865,Z -53.525,A -90.000,B 90.000,C 0.000} C_DIS
LIN {X -9.373,Y -27.870,Z -53.528,A -90.000,B 90.000,C 0.000} C_DIS
LIN {X -9.171,Y -27.873,Z -53.539,A -90.000,B 90.000,C 0.000} C_DIS
LIN {X -8.164,Y -27.914,Z -53.621,A -90.000,B 90.000,C 0.000} C_DIS
LIN {X -7.484,Y -27.949,Z -53.680,A -90.000,B 90.000,C 0.000} C_DIS
LIN {X -7.044,Y -27.968,Z -53.726,A -90.000,B 90.000,C 0.000} C_DIS
LIN {X -6.847,Y -27.975,Z -53.752,A -90.000,B 90.000,C 0.000} C_DIS
LIN {X -6.708,Y -27.977,Z -53.774,A -90.000,B 90.000,C 0.000} C_DIS
LIN {X -6.567,Y -27.978,Z -53.796,A -90.000,B 90.000,C 0.000} C_DIS
LIN {X -6.196,Y -27.987,Z -53.858,A -90.000,B 90.000,C 0.000} C_DIS
LIN {X -5.879,Y -28.003,Z -53.920,A -90.000,B 90.000,C 0.000} C_DIS
LIN {X -4.355,Y -28.073,Z -54.230,A -90.000,B 90.000,C 0.000} C_DIS
LIN {X -3.772,Y -28.078,Z -54.369,A -90.000,B 90.000,C 0.000} C_DIS
LIN {X -3.571,Y -28.085,Z -54.422,A -90.000,B 90.000,C 0.000} C_DIS
LIN {X -2.864,Y -28.099,Z -54.618,A -90.000,B 90.000,C 0.000} C_DIS
LIN {X -1.597,Y -28.143,Z -54.954,A -90.000,B 90.000,C 0.000} C_DIS
LIN {X -0.977,Y -28.144,Z -55.137,A -90.000,B 90.000,C 0.000} C_DIS
LIN {X 0.012,Y -28.161,Z -55.419,A -90.000,B 90.000,C 0.000} C_DIS
LIN {X 0.536,Y -28.168,Z -55.568,A -90.000,B 90.000,C 0.000} C_DIS
LIN {X 0.915,Y -28.168,Z -55.680,A -90.000,B 90.000,C 0.000} C_DIS
LIN {X 1.053,Y -28.171,Z -55.719,A -90.000,B 90.000,C 0.000} C_DIS
LIN {X 1.679,Y -28.172,Z -55.885,A -90.000,B 90.000,C 0.000} C_DIS
LIN {X 2.772,Y -28.170,Z -56.166,A -90.000,B 90.000,C 0.000} C_DIS
LIN {X 3.384,Y -28.183,Z -56.313,A -90.000,B 90.000,C 0.000} C_DIS
LIN {X 4.180,Y -28.168,Z -56.458,A -90.000,B 90.000,C 0.000} C_DIS
LIN {X 4.782,Y -28.176,Z -56.554,A -90.000,B 90.000,C 0.000} C_DIS
LIN {X 5.118,Y -28.185,Z -56.602,A -90.000,B 90.000,C 0.000} C_DIS
LIN {X 5.519,Y -28.180,Z -56.636,A -90.000,B 90.000,C 0.000} C_DIS
LIN {X 6.195,Y -28.194,Z -56.679,A -90.000,B 90.000,C 0.000} C_DIS
LIN {X 6.359,Y -28.199,Z -56.688,A -90.000,B 90.000,C 0.000} C_DIS
LIN {X 6.837,Y -28.200,Z -56.695,A -90.000,B 90.000,C 0.000} C_DIS
LIN {X 7.088,Y -28.206,Z -56.693,A -90.000,B 90.000,C 0.000} C_DIS
LIN {X 7.609,Y -28.216,Z -56.685,A -90.000,B 90.000,C 0.000} C_DIS
LIN {X 7.964,Y -28.216,Z -56.666,A -90.000,B 90.000,C 0.000} C_DIS
LIN {X 8.604,Y -28.229,Z -56.622,A -90.000,B 90.000,C 0.000} C_DIS
LIN {X 9.331,Y -28.233,Z -56.559,A -90.000,B 90.000,C 0.000} C_DIS
LIN {X 9.798,Y -28.233,Z -56.521,A -90.000,B 90.000,C 0.000} C_DIS
LIN {X 10.601,Y -28.238,Z -56.468,A -90.000,B 90.000,C 0.000} C_DIS
LIN {X 10.818,Y -28.238,Z -56.454,A -90.000,B 90.000,C 0.000} C_DIS
LIN {X 11.167,Y -28.221,Z -56.435,A -90.000,B 90.000,C 0.000} C_DIS
LIN {X 11.374,Y -28.213,Z -56.426,A -90.000,B 90.000,C 0.000} C_DIS
LIN {X 11.880,Y -28.195,Z -56.408,A -90.000,B 90.000,C 0.000} C_DIS
LIN {X 12.005,Y -28.185,Z -56.395,A -90.000,B 90.000,C 0.000} C_DIS
LIN {X 12.156,Y -28.177,Z -56.383,A -90.000,B 90.000,C 0.000} C_DIS
LIN {X 12.209,Y -28.176,Z -56.379,A -90.000,B 90.000,C 0.000} C_DIS
LIN {X 12.733,Y -28.139,Z -56.360,A -90.000,B 90.000,C 0.000} C_DIS
LIN {X 12.885,Y -28.123,Z -56.348,A -90.000,B 90.000,C 0.000} C_DIS
LIN {X 13.249,Y -28.090,Z -56.325,A -90.000,B 90.000,C 0.000} C_DIS
LIN {X 13.324,Y -28.081,Z -56.314,A -90.000,B 90.000,C 0.000} C_DIS
LIN {X 13.599,Y -28.046,Z -56.279,A -90.000,B 90.000,C 0.000} C_DIS
LIN {X 13.779,Y -28.027,Z -56.261,A -90.000,B 90.000,C 0.000} C_DIS
LIN {X 13.808,Y -28.025,Z -56.259,A -90.000,B 90.000,C 0.000} C_DIS
LIN {X 14.021,Y -27.995,Z -56.229,A -90.000,B 90.000,C 0.000} C_DIS
LIN {X 14.140,Y -27.981,Z -56.215,A -90.000,B 90.000,C 0.000} C_DIS
LIN {X 14.590,Y -27.939,Z -56.181,A -90.000,B 90.000,C 0.000} C_DIS
LIN {X 14.778,Y -27.915,Z -56.157,A -90.000,B 90.000,C 0.000} C_DIS
LIN {X 14.941,Y -27.898,Z -56.141,A -90.000,B 90.000,C 0.000} C_DIS
LIN {X 15.141,Y -27.884,Z -56.127,A -90.000,B 90.000,C 0.000} C_DIS
LIN {X 15.423,Y -27.868,Z -56.105,A -90.000,B 90.000,C 0.000} C_DIS
LIN {X 15.852,Y -27.858,Z -56.089,A -90.000,B 90.000,C 0.000} C_DIS
LIN {X 16.032,Y -27.845,Z -56.078,A -90.000,B 90.000,C 0.000} C_DIS
LIN {X 16.193,Y -27.837,Z -56.073,A -90.000,B 90.000,C 0.000} C_DIS
LIN {X 16.616,Y -27.828,Z -56.073,A -90.000,B 90.000,C 0.000} C_DIS
LIN {X 16.732,Y -27.828,Z -56.075,A -90.000,B 90.000,C 0.000} C_DIS
LIN {X 16.845,Y -27.833,Z -56.079,A -90.000,B 90.000,C 0.000} C_DIS
LIN {X 17.233,Y -27.835,Z -56.110,A -90.000,B 90.000,C 0.000} C_DIS
LIN {X 17.392,Y -27.830,Z -56.121,A -90.000,B 90.000,C 0.000} C_DIS
LIN {X 17.859,Y -27.829,Z -56.167,A -90.000,B 90.000,C 0.000} C_DIS
LIN {X 17.909,Y -27.830,Z -56.173,A -90.000,B 90.000,C 0.000} C_DIS
LIN {X 18.344,Y -27.829,Z -56.267,A -90.000,B 90.000,C 0.000} C_DIS
LIN {X 18.402,Y -27.827,Z -56.281,A -90.000,B 90.000,C 0.000} C_DIS
LIN {X 18.919,Y -27.841,Z -56.407,A -90.000,B 90.000,C 0.000} C_DIS
LIN {X 19.079,Y -27.835,Z -56.456,A -90.000,B 90.000,C 0.000} C_DIS
LIN {X 19.239,Y -27.782,Z -56.460,A -90.000,B 90.000,C 0.000} C_DIS
LIN {X 19.375,Y -27.739,Z -56.466,A -90.000,B 90.000,C 0.000} C_DIS
LIN {X 19.602,Y -27.664,Z -56.490,A -90.000,B 90.000,C 0.000} C_DIS
LIN {X 19.749,Y -27.697,Z -56.396,A -90.000,B 90.000,C 0.000} C_DIS
LIN {X 19.989,Y -27.756,Z -56.258,A -90.000,B 90.000,C 0.000} C_DIS
LIN {X 20.151,Y -27.801,Z -56.164,A -90.000,B 90.000,C 0.000} C_DIS
LIN {X 20.286,Y -27.839,Z -56.096,A -90.000,B 90.000,C 0.000} C_DIS
LIN {X 20.504,Y -27.906,Z -55.996,A -90.000,B 90.000,C 0.000} C_DIS
LIN {X 20.735,Y -27.979,Z -55.894,A -90.000,B 90.000,C 0.000} C_DIS
LIN {X 20.843,Y -28.016,Z -55.852,A -90.000,B 90.000,C 0.000} C_DIS
LIN {X 20.956,Y -28.056,Z -55.810,A -90.000,B 90.000,C 0.000} C_DIS
LIN {X 21.245,Y -28.113,Z -55.588,A -90.000,B 90.000,C 0.000} C_DIS
LIN {X 21.362,Y -28.062,Z -55.347,A -90.000,B 90.000,C 0.000} C_DIS
LIN {X 21.386,Y -28.051,Z -55.305,A -90.000,B 90.000,C 0.000} C_DIS
LIN {X 21.479,Y -28.017,Z -55.143,A -90.000,B 90.000,C 0.000} C_DIS
LIN {X 21.606,Y -27.972,Z -54.926,A -90.000,B 90.000,C 0.000} C_DIS
LIN {X 21.666,Y -27.948,Z -54.841,A -90.000,B 90.000,C 0.000} C_DIS
LIN {X 21.718,Y -27.931,Z -54.771,A -90.000,B 90.000,C 0.000} C_DIS
LIN {X 21.781,Y -27.928,Z -54.655,A -90.000,B 90.000,C 0.000} C_DIS
LIN {X 21.939,Y -27.907,Z -54.391,A -90.000,B 90.000,C 0.000} C_DIS
LIN {X 22.029,Y -27.896,Z -54.268,A -90.000,B 90.000,C 0.000} C_DIS
LIN {X 22.146,Y -27.879,Z -54.100,A -90.000,B 90.000,C 0.000} C_DIS
LIN {X 22.235,Y -27.870,Z -53.980,A -90.000,B 90.000,C 0.000} C_DIS
LIN {X 22.477,Y -27.838,Z -53.687,A -90.000,B 90.000,C 0.000} C_DIS
LIN {X 22.547,Y -27.831,Z -53.608,A -90.000,B 90.000,C 0.000} C_DIS
LIN {X 22.661,Y -27.864,Z -53.422,A -90.000,B 90.000,C 0.000} C_DIS
LIN {X 22.895,Y -27.917,Z -53.076,A -90.000,B 90.000,C 0.000} C_DIS
LIN {X 23.015,Y -27.948,Z -52.896,A -90.000,B 90.000,C 0.000} C_DIS
LIN {X 23.123,Y -27.978,Z -52.753,A -90.000,B 90.000,C 0.000} C_DIS
LIN {X 23.370,Y -28.040,Z -52.449,A -90.000,B 90.000,C 0.000} C_DIS
LIN {X 23.478,Y -28.070,Z -52.321,A -90.000,B 90.000,C 0.000} C_DIS
LIN {X 23.591,Y -28.100,Z -52.193,A -90.000,B 90.000,C 0.000} C_DIS
LIN {X 23.873,Y -28.180,Z -51.894,A -90.000,B 90.000,C 0.000} C_DIS
LIN {X 23.897,Y -28.187,Z -51.869,A -90.000,B 90.000,C 0.000} C_DIS
LIN {X 23.927,Y -28.178,Z -51.757,A -90.000,B 90.000,C 0.000} C_DIS
LIN {X 24.022,Y -28.155,Z -51.429,A -90.000,B 90.000,C 0.000} C_DIS
LIN {X 24.037,Y -28.150,Z -51.383,A -90.000,B 90.000,C 0.000} C_DIS
LIN {X 24.128,Y -28.124,Z -51.129,A -90.000,B 90.000,C 0.000} C_DIS
LIN {X 24.172,Y -28.110,Z -51.002,A -90.000,B 90.000,C 0.000} C_DIS
LIN {X 24.244,Y -28.092,Z -50.821,A -90.000,B 90.000,C 0.000} C_DIS
LIN {X 24.312,Y -28.079,Z -50.663,A -90.000,B 90.000,C 0.000} C_DIS
LIN {X 24.446,Y -28.045,Z -50.381,A -90.000,B 90.000,C 0.000} C_DIS
LIN {X 24.557,Y -28.022,Z -50.162,A -90.000,B 90.000,C 0.000} C_DIS
LIN {X 24.696,Y -27.998,Z -49.888,A -90.000,B 90.000,C 0.000} C_DIS
LIN {X 24.756,Y -27.990,Z -49.774,A -90.000,B 90.000,C 0.000} C_DIS
LIN {X 24.988,Y -27.950,Z -49.371,A -90.000,B 90.000,C 0.000} C_DIS
LIN {X 25.069,Y -27.940,Z -49.239,A -90.000,B 90.000,C 0.000} C_DIS
LIN {X 25.271,Y -27.908,Z -48.925,A -90.000,B 90.000,C 0.000} C_DIS
LIN {X 25.401,Y -27.883,Z -48.734,A -90.000,B 90.000,C 0.000} C_DIS
LIN {X 25.537,Y -27.863,Z -48.549,A -90.000,B 90.000,C 0.000} C_DIS
LIN {X 25.875,Y -27.816,Z -48.106,A -90.000,B 90.000,C 0.000} C_DIS
LIN {X 25.985,Y -27.797,Z -47.984,A -90.000,B 90.000,C 0.000} C_DIS
LIN {X 26.115,Y -27.785,Z -47.820,A -90.000,B 90.000,C 0.000} C_DIS
LIN {X 26.216,Y -27.770,Z -47.711,A -90.000,B 90.000,C 0.000} C_DIS
LIN {X 26.442,Y -27.748,Z -47.480,A -90.000,B 90.000,C 0.000} C_DIS
LIN {X 26.605,Y -27.734,Z -47.315,A -90.000,B 90.000,C 0.000} C_DIS
LIN {X 26.929,Y -27.695,Z -47.022,A -90.000,B 90.000,C 0.000} C_DIS
LIN {X 27.146,Y -27.675,Z -46.815,A -90.000,B 90.000,C 0.000} C_DIS
LIN {X 27.179,Y -27.671,Z -46.787,A -90.000,B 90.000,C 0.000} C_DIS
LIN {X 27.246,Y -27.663,Z -46.730,A -90.000,B 90.000,C 0.000} C_DIS
LIN {X 27.351,Y -27.653,Z -46.643,A -90.000,B 90.000,C 0.000} C_DIS
LIN {X 27.459,Y -27.646,Z -46.556,A -90.000,B 90.000,C 0.000} C_DIS
LIN {X 27.709,Y -27.620,Z -46.376,A -90.000,B 90.000,C 0.000} C_DIS
LIN {X 28.067,Y -27.597,Z -46.133,A -90.000,B 90.000,C 0.000} C_DIS
LIN {X 28.280,Y -27.577,Z -46.006,A -90.000,B 90.000,C 0.000} C_DIS
LIN {X 28.609,Y -27.562,Z -45.820,A -90.000,B 90.000,C 0.000} C_DIS
LIN {X 28.969,Y -27.526,Z -45.642,A -90.000,B 90.000,C 0.000} C_DIS
LIN {X 29.272,Y -27.509,Z -45.482,A -90.000,B 90.000,C 0.000} C_DIS
LIN {X 29.398,Y -27.503,Z -45.417,A -90.000,B 90.000,C 0.000} C_DIS
LIN {X 29.547,Y -27.495,Z -45.348,A -90.000,B 90.000,C 0.000} C_DIS
LIN {X 29.807,Y -27.487,Z -45.232,A -90.000,B 90.000,C 0.000} C_DIS
LIN {X 30.147,Y -27.468,Z -45.105,A -90.000,B 90.000,C 0.000} C_DIS
LIN {X 30.437,Y -27.460,Z -45.001,A -90.000,B 90.000,C 0.000} C_DIS
LIN {X 30.640,Y -27.450,Z -44.942,A -90.000,B 90.000,C 0.000} C_DIS
LIN {X 30.879,Y -27.443,Z -44.875,A -90.000,B 90.000,C 0.000} C_DIS
LIN {X 31.297,Y -27.424,Z -44.789,A -90.000,B 90.000,C 0.000} C_DIS
LIN {X 31.768,Y -27.407,Z -44.694,A -90.000,B 90.000,C 0.000} C_DIS
LIN {X 31.944,Y -27.401,Z -44.660,A -90.000,B 90.000,C 0.000} C_DIS
LIN {X 32.195,Y -27.392,Z -44.623,A -90.000,B 90.000,C 0.000} C_DIS
LIN {X 32.416,Y -27.387,Z -44.591,A -90.000,B 90.000,C 0.000} C_DIS
LIN {X 32.852,Y -27.378,Z -44.538,A -90.000,B 90.000,C 0.000} C_DIS
LIN {X 33.246,Y -27.374,Z -44.492,A -90.000,B 90.000,C 0.000} C_DIS
LIN {X 33.338,Y -27.374,Z -44.483,A -90.000,B 90.000,C 0.000} C_DIS
LIN {X 33.989,Y -27.367,Z -44.456,A -90.000,B 90.000,C 0.000} C_DIS
LIN {X 34.388,Y -27.366,Z -44.444,A -90.000,B 90.000,C 0.000} C_DIS
LIN {X 34.529,Y -27.365,Z -44.441,A -90.000,B 90.000,C 0.000} C_DIS
LIN {X 34.827,Y -27.364,Z -44.437,A -90.000,B 90.000,C 0.000} C_DIS
LIN {X 34.969,Y -27.362,Z -44.440,A -90.000,B 90.000,C 0.000} C_DIS
LIN {X 35.363,Y -27.361,Z -44.433,A -90.000,B 90.000,C 0.000} C_DIS
LIN {X 35.679,Y -27.365,Z -44.430,A -90.000,B 90.000,C 0.000} C_DIS
LIN {X 36.018,Y -27.369,Z -44.434,A -90.000,B 90.000,C 0.000} C_DIS
LIN {X 36.445,Y -27.386,Z -44.404,A -90.000,B 90.000,C 0.000} C_DIS
LIN {X 36.511,Y -27.388,Z -44.401,A -90.000,B 90.000,C 0.000} C_DIS
LIN {X 36.792,Y -27.411,Z -44.349,A -90.000,B 90.000,C 0.000} C_DIS
LIN {X 37.036,Y -27.433,Z -44.305,A -90.000,B 90.000,C 0.000} C_DIS
LIN {X 37.365,Y -27.474,Z -44.225,A -90.000,B 90.000,C 0.000} C_DIS
LIN {X 37.844,Y -27.541,Z -44.114,A -90.000,B 90.000,C 0.000} C_DIS
LIN {X 38.152,Y -27.590,Z -44.046,A -90.000,B 90.000,C 0.000} C_DIS
LIN {X 38.434,Y -27.626,Z -43.978,A -90.000,B 90.000,C 0.000} C_DIS
LIN {X 38.630,Y -27.654,Z -43.929,A -90.000,B 90.000,C 0.000} C_DIS
LIN {X 39.090,Y -27.683,Z -43.787,A -90.000,B 90.000,C 0.000} C_DIS
LIN {X 40.226,Y -27.699,Z -43.394,A -90.000,B 90.000,C 0.000} C_DIS
LIN {X 40.643,Y -27.696,Z -43.262,A -90.000,B 90.000,C 0.000} C_DIS
LIN {X 40.709,Y -27.693,Z -43.245,A -90.000,B 90.000,C 0.000} C_DIS
LIN {X 41.723,Y -27.666,Z -42.949,A -90.000,B 90.000,C 0.000} C_DIS
LIN {X 42.277,Y -27.657,Z -42.792,A -90.000,B 90.000,C 0.000} C_DIS
LIN {X 42.334,Y -27.657,Z -42.777,A -90.000,B 90.000,C 0.000} C_DIS
LIN {X 42.784,Y -27.649,Z -42.685,A -90.000,B 90.000,C 0.000} C_DIS
LIN {X 43.023,Y -27.649,Z -42.640,A -90.000,B 90.000,C 0.000} C_DIS
LIN {X 43.521,Y -27.640,Z -42.562,A -90.000,B 90.000,C 0.000} C_DIS
LIN {X 43.966,Y -27.630,Z -42.498,A -90.000,B 90.000,C 0.000} C_DIS
LIN {X 44.606,Y -27.589,Z -42.448,A -90.000,B 90.000,C 0.000} C_DIS
LIN {X 44.708,Y -27.586,Z -42.441,A -90.000,B 90.000,C 0.000} C_DIS
LIN {X 45.023,Y -27.581,Z -42.424,A -90.000,B 90.000,C 0.000} C_DIS
LIN {X 45.423,Y -27.571,Z -42.411,A -90.000,B 90.000,C 0.000} C_DIS
LIN {X 45.781,Y -27.570,Z -42.406,A -90.000,B 90.000,C 0.000} C_DIS
LIN {X 46.400,Y -27.543,Z -42.448,A -90.000,B 90.000,C 0.000} C_DIS
LIN {X 46.541,Y -27.536,Z -42.460,A -90.000,B 90.000,C 0.000} C_DIS
LIN {X 46.671,Y -27.533,Z -42.473,A -90.000,B 90.000,C 0.000} C_DIS
LIN {X 47.126,Y -27.526,Z -42.528,A -90.000,B 90.000,C 0.000} C_DIS
LIN {X 47.984,Y -27.503,Z -42.653,A -90.000,B 90.000,C 0.000} C_DIS
LIN {X 48.374,Y -27.481,Z -42.737,A -90.000,B 90.000,C 0.000} C_DIS
LIN {X 48.636,Y -27.473,Z -42.797,A -90.000,B 90.000,C 0.000} C_DIS
LIN {X 49.118,Y -27.466,Z -42.912,A -90.000,B 90.000,C 0.000} C_DIS
LIN {X 49.662,Y -27.468,Z -43.046,A -90.000,B 90.000,C 0.000} C_DIS
LIN {X 50.009,Y -27.461,Z -43.157,A -90.000,B 90.000,C 0.000} C_DIS
LIN {X 50.405,Y -27.456,Z -43.295,A -90.000,B 90.000,C 0.000} C_DIS
LIN {X 51.010,Y -27.443,Z -43.527,A -90.000,B 90.000,C 0.000} C_DIS
LIN {X 51.492,Y -27.437,Z -43.715,A -90.000,B 90.000,C 0.000} C_DIS
LIN {X 51.614,Y -27.437,Z -43.764,A -90.000,B 90.000,C 0.000} C_DIS
LIN {X 52.345,Y -27.423,Z -44.088,A -90.000,B 90.000,C 0.000} C_DIS
LIN {X 52.545,Y -27.419,Z -44.183,A -90.000,B 90.000,C 0.000} C_DIS
LIN {X 52.987,Y -27.419,Z -44.398,A -90.000,B 90.000,C 0.000} C_DIS
LIN {X 53.415,Y -27.419,Z -44.615,A -90.000,B 90.000,C 0.000} C_DIS
LIN {X 53.601,Y -27.414,Z -44.726,A -90.000,B 90.000,C 0.000} C_DIS
LIN {X 54.428,Y -27.401,Z -45.224,A -90.000,B 90.000,C 0.000} C_DIS
LIN {X 55.640,Y -27.381,Z -45.978,A -90.000,B 90.000,C 0.000} C_DIS
LIN {X 56.062,Y -27.383,Z -46.243,A -90.000,B 90.000,C 0.000} C_DIS
LIN {X 56.432,Y -27.393,Z -46.486,A -90.000,B 90.000,C 0.000} C_DIS
LIN {X 56.915,Y -27.392,Z -46.868,A -90.000,B 90.000,C 0.000} C_DIS
LIN {X 58.413,Y -27.386,Z -48.073,A -90.000,B 90.000,C 0.000} C_DIS
LIN {X 58.892,Y -27.383,Z -48.469,A -90.000,B 90.000,C 0.000} C_DIS
LIN {X 59.082,Y -27.386,Z -48.628,A -90.000,B 90.000,C 0.000} C_DIS
LIN {X 61.166,Y -27.374,Z -50.582,A -90.000,B 90.000,C 0.000} C_DIS
LIN {X 62.237,Y -27.373,Z -51.610,A -90.000,B 90.000,C 0.000} C_DIS
LIN {X 63.161,Y -27.370,Z -52.500,A -90.000,B 90.000,C 0.000} C_DIS
LIN {X 64.070,Y -27.373,Z -53.305,A -90.000,B 90.000,C 0.000} C_DIS
LIN {X 64.999,Y -27.374,Z -54.142,A -90.000,B 90.000,C 0.000} C_DIS
LIN {X 65.223,Y -27.379,Z -54.313,A -90.000,B 90.000,C 0.000} C_DIS
LIN {X 66.289,Y -27.386,Z -55.123,A -90.000,B 90.000,C 0.000} C_DIS
LIN {X 66.881,Y -27.391,Z -55.557,A -90.000,B 90.000,C 0.000} C_DIS
LIN {X 67.888,Y -27.403,Z -56.262,A -90.000,B 90.000,C 0.000} C_DIS
LIN {X 69.005,Y -27.422,Z -57.013,A -90.000,B 90.000,C 0.000} C_DIS
LIN {X 70.557,Y -27.446,Z -58.109,A -90.000,B 90.000,C 0.000} C_DIS
LIN {X 71.043,Y -27.458,Z -58.441,A -90.000,B 90.000,C 0.000} C_DIS
LIN {X 71.548,Y -27.456,Z -58.837,A -90.000,B 90.000,C 0.000} C_DIS
LIN {X 72.017,Y -27.466,Z -59.211,A -90.000,B 90.000,C 0.000} C_DIS
LIN {X 72.898,Y -27.489,Z -59.921,A -90.000,B 90.000,C 0.000} C_DIS
LIN {X 73.107,Y -27.496,Z -60.087,A -90.000,B 90.000,C 0.000} C_DIS
LIN {X 73.202,Y -27.495,Z -60.175,A -90.000,B 90.000,C 0.000} C_DIS
LIN {X 73.599,Y -27.490,Z -60.558,A -90.000,B 90.000,C 0.000} C_DIS
LIN {X 73.679,Y -27.493,Z -60.638,A -90.000,B 90.000,C 0.000} C_DIS
LIN {X 74.188,Y -27.509,Z -61.165,A -90.000,B 90.000,C 0.000} C_DIS
LIN {X 74.727,Y -27.524,Z -61.736,A -90.000,B 90.000,C 0.000} C_DIS
LIN {X 74.765,Y -27.524,Z -61.778,A -90.000,B 90.000,C 0.000} C_DIS
LIN {X 74.892,Y -27.527,Z -61.918,A -90.000,B 90.000,C 0.000} C_DIS
LIN {X 75.192,Y -27.524,Z -62.275,A -90.000,B 90.000,C 0.000} C_DIS
LIN {X 75.417,Y -27.518,Z -62.560,A -90.000,B 90.000,C 0.000} C_DIS
LIN {X 75.853,Y -27.527,Z -63.127,A -90.000,B 90.000,C 0.000} C_DIS
LIN {X 76.358,Y -27.531,Z -63.794,A -90.000,B 90.000,C 0.000} C_DIS
LIN {X 76.619,Y -27.523,Z -64.179,A -90.000,B 90.000,C 0.000} C_DIS
LIN {X 76.891,Y -27.521,Z -64.587,A -90.000,B 90.000,C 0.000} C_DIS
LIN {X 77.493,Y -27.532,Z -65.509,A -90.000,B 90.000,C 0.000} C_DIS
LIN {X 77.589,Y -27.531,Z -65.657,A -90.000,B 90.000,C 0.000} C_DIS
LIN {X 77.803,Y -27.522,Z -66.002,A -90.000,B 90.000,C 0.000} C_DIS
LIN {X 78.177,Y -27.519,Z -66.619,A -90.000,B 90.000,C 0.000} C_DIS
LIN {X 78.408,Y -27.515,Z -66.976,A -90.000,B 90.000,C 0.000} C_DIS
LIN {X 78.448,Y -27.490,Z -67.017,A -90.000,B 90.000,C 0.000} C_DIS
LIN {X 78.492,Y -27.488,Z -66.781,A -90.000,B 90.000,C 0.000} C_DIS
LIN {X 78.566,Y -27.496,Z -66.415,A -90.000,B 90.000,C 0.000} C_DIS
LIN {X 78.619,Y -27.502,Z -66.158,A -90.000,B 90.000,C 0.000} C_DIS
LIN {X 79.071,Y -27.498,Z -64.443,A -90.000,B 90.000,C 0.000} C_DIS
LIN {X 79.177,Y -27.511,Z -64.054,A -90.000,B 90.000,C 0.000} C_DIS
LIN {X 79.220,Y -27.514,Z -63.914,A -90.000,B 90.000,C 0.000} C_DIS
LIN {X 79.344,Y -27.520,Z -63.543,A -90.000,B 90.000,C 0.000} C_DIS
LIN {X 79.555,Y -27.532,Z -62.912,A -90.000,B 90.000,C 0.000} C_DIS
LIN {X 79.932,Y -27.547,Z -61.833,A -90.000,B 90.000,C 0.000} C_DIS
LIN {X 80.528,Y -27.573,Z -60.219,A -90.000,B 90.000,C 0.000} C_DIS
LIN {X 80.606,Y -27.579,Z -60.009,A -90.000,B 90.000,C 0.000} C_DIS
LIN {X 80.754,Y -27.588,Z -59.626,A -90.000,B 90.000,C 0.000} C_DIS
LIN {X 81.125,Y -27.583,Z -58.754,A -90.000,B 90.000,C 0.000} C_DIS
LIN {X 81.578,Y -27.622,Z -57.497,A -90.000,B 90.000,C 0.000} C_DIS
LIN {X 82.437,Y -27.668,Z -55.488,A -90.000,B 90.000,C 0.000} C_DIS
LIN {X 82.627,Y -27.669,Z -55.056,A -90.000,B 90.000,C 0.000} C_DIS
LIN {X 83.498,Y -27.614,Z -53.311,A -90.000,B 90.000,C 0.000} C_DIS
LIN {X 83.638,Y -27.612,Z -53.033,A -90.000,B 90.000,C 0.000} C_DIS
LIN {X 83.725,Y -27.607,Z -52.878,A -90.000,B 90.000,C 0.000} C_DIS
LIN {X 84.158,Y -27.571,Z -52.138,A -90.000,B 90.000,C 0.000} C_DIS
LIN {X 84.805,Y -27.528,Z -51.083,A -90.000,B 90.000,C 0.000} C_DIS
LIN {X 84.929,Y -27.525,Z -50.887,A -90.000,B 90.000,C 0.000} C_DIS
LIN {X 85.043,Y -27.519,Z -50.717,A -90.000,B 90.000,C 0.000} C_DIS
LIN {X 85.635,Y -27.478,Z -49.899,A -90.000,B 90.000,C 0.000} C_DIS
LIN {X 86.064,Y -27.458,Z -49.313,A -90.000,B 90.000,C 0.000} C_DIS
LIN {X 86.348,Y -27.451,Z -48.928,A -90.000,B 90.000,C 0.000} C_DIS
LIN {X 86.694,Y -27.434,Z -48.518,A -90.000,B 90.000,C 0.000} C_DIS
LIN {X 87.043,Y -27.417,Z -48.110,A -90.000,B 90.000,C 0.000} C_DIS
LIN {X 87.759,Y -27.389,Z -47.324,A -90.000,B 90.000,C 0.000} C_DIS
LIN {X 88.115,Y -27.382,Z -46.935,A -90.000,B 90.000,C 0.000} C_DIS
LIN {X 88.342,Y -27.374,Z -46.717,A -90.000,B 90.000,C 0.000} C_DIS
LIN {X 88.725,Y -27.361,Z -46.366,A -90.000,B 90.000,C 0.000} C_DIS
LIN {X 89.544,Y -27.338,Z -45.626,A -90.000,B 90.000,C 0.000} C_DIS
LIN {X 89.868,Y -27.334,Z -45.334,A -90.000,B 90.000,C 0.000} C_DIS
LIN {X 90.066,Y -27.331,Z -45.160,A -90.000,B 90.000,C 0.000} C_DIS
LIN {X 90.916,Y -27.319,Z -44.499,A -90.000,B 90.000,C 0.000} C_DIS
LIN {X 91.730,Y -27.312,Z -43.866,A -90.000,B 90.000,C 0.000} C_DIS
LIN {X 92.155,Y -27.311,Z -43.556,A -90.000,B 90.000,C 0.000} C_DIS
LIN {X 93.797,Y -27.308,Z -42.409,A -90.000,B 90.000,C 0.000} C_DIS
LIN {X 94.526,Y -27.315,Z -41.947,A -90.000,B 90.000,C 0.000} C_DIS
LIN {X 94.549,Y -27.318,Z -41.933,A -90.000,B 90.000,C 0.000} C_DIS
LIN {X 94.821,Y -27.318,Z -41.760,A -90.000,B 90.000,C 0.000} C_DIS
LIN {X 95.417,Y -27.308,Z -41.383,A -90.000,B 90.000,C 0.000} C_DIS
LIN {X 95.600,Y -27.304,Z -41.268,A -90.000,B 90.000,C 0.000} C_DIS
LIN {X 95.601,Y -29.847,Z -41.268,A -90.000,B 90.000,C 0.000} C_DIS
LIN {X 95.598,Y -27.306,Z -41.269,A -90.000,B 90.000,C 0.000} C_DIS
LIN {X 95.610,Y -27.306,Z -41.262,A -90.000,B 90.000,C 0.000} C_DIS
LIN {X 95.662,Y -27.307,Z -41.232,A -90.000,B 90.000,C 0.000} C_DIS
LIN {X 95.766,Y -27.308,Z -41.178,A -90.000,B 90.000,C 0.000} C_DIS
LIN {X 95.838,Y -27.308,Z -41.136,A -90.000,B 90.000,C 0.000} C_DIS
LIN {X 95.838,Y -60.000,Z -41.136,A -90.000,B 90.000,C 0.000} C_DIS
LIN {X 117.202,Y -60.000,Z -45.935,A -90.000,B 90.000,C 0.000} C_DIS
LIN {X 117.202,Y -27.308,Z -45.935,A -90.000,B 90.000,C 0.000} C_DIS
LIN {X 117.121,Y -27.308,Z -46.207,A -90.000,B 90.000,C 0.000} C_DIS
LIN {X 117.121,Y -60.000,Z -46.207,A -90.000,B 90.000,C 0.000} C_DIS
LIN {X -40.964,Y -60.000,Z -52.963,A -90.000,B 90.000,C 0.000} C_DIS
LIN {X -40.964,Y -27.308,Z -52.963,A -90.000,B 90.000,C 0.000} C_DIS
LIN {X -39.615,Y -27.371,Z -53.239,A -90.000,B 90.000,C 0.000} C_DIS
LIN {X -39.032,Y -27.399,Z -53.360,A -90.000,B 90.000,C 0.000} C_DIS
LIN {X -38.416,Y -27.419,Z -53.494,A -90.000,B 90.000,C 0.000} C_DIS
LIN {X -37.067,Y -27.464,Z -53.792,A -90.000,B 90.000,C 0.000} C_DIS
LIN {X -36.082,Y -27.495,Z -54.013,A -90.000,B 90.000,C 0.000} C_DIS
LIN {X -35.555,Y -27.509,Z -54.134,A -90.000,B 90.000,C 0.000} C_DIS
LIN {X -34.661,Y -27.516,Z -54.324,A -90.000,B 90.000,C 0.000} C_DIS
LIN {X -34.109,Y -27.507,Z -54.415,A -90.000,B 90.000,C 0.000} C_DIS
LIN {X -32.694,Y -27.455,Z -54.597,A -90.000,B 90.000,C 0.000} C_DIS
LIN {X -32.004,Y -27.425,Z -54.689,A -90.000,B 90.000,C 0.000} C_DIS
LIN {X -31.071,Y -27.392,Z -54.825,A -90.000,B 90.000,C 0.000} C_DIS
LIN {X -29.554,Y -27.323,Z -55.057,A -90.000,B 90.000,C 0.000} C_DIS
LIN {X -29.203,Y -27.308,Z -55.110,A -90.000,B 90.000,C 0.000} C_DIS
LIN {X -29.203,Y -60.000,Z -55.110,A -90.000,B 90.000,C 0.000} C_DIS
LIN {X -76.950,Y -60.000,Z -52.648,A -90.000,B 90.000,C 0.000} C_DIS
LIN {X -76.950,Y -27.308,Z -52.648,A -90.000,B 90.000,C 0.000} C_DIS
LIN {X -76.627,Y -27.386,Z -52.832,A -90.000,B 90.000,C 0.000} C_DIS
LIN {X -76.264,Y -27.478,Z -53.056,A -90.000,B 90.000,C 0.000} C_DIS
LIN {X -76.128,Y -27.515,Z -53.147,A -90.000,B 90.000,C 0.000} C_DIS
LIN {X -75.759,Y -27.610,Z -53.377,A -90.000,B 90.000,C 0.000} C_DIS
LIN {X -75.077,Y -27.784,Z -53.788,A -90.000,B 90.000,C 0.000} C_DIS
LIN {X -74.876,Y -27.837,Z -53.911,A -90.000,B 90.000,C 0.000} C_DIS
LIN {X -74.643,Y -27.903,Z -54.065,A -90.000,B 90.000,C 0.000} C_DIS
LIN {X -74.434,Y -27.951,Z -54.165,A -90.000,B 90.000,C 0.000} C_DIS
LIN {X -74.254,Y -27.980,Z -54.205,A -90.000,B 90.000,C 0.000} C_DIS
LIN {X -74.173,Y -27.991,Z -54.218,A -90.000,B 90.000,C 0.000} C_DIS
LIN {X -73.530,Y -28.062,Z -54.253,A -90.000,B 90.000,C 0.000} C_DIS
LIN {X -72.694,Y -28.122,Z -54.116,A -90.000,B 90.000,C 0.000} C_DIS
LIN {X -71.804,Y -28.185,Z -53.983,A -90.000,B 90.000,C 0.000} C_DIS
LIN {X -71.322,Y -28.210,Z -53.867,A -90.000,B 90.000,C 0.000} C_DIS
LIN {X -71.234,Y -28.215,Z -53.846,A -90.000,B 90.000,C 0.000} C_DIS
LIN {X -70.425,Y -28.269,Z -53.672,A -90.000,B 90.000,C 0.000} C_DIS
LIN {X -69.712,Y -28.309,Z -53.487,A -90.000,B 90.000,C 0.000} C_DIS
LIN {X -69.174,Y -28.327,Z -53.310,A -90.000,B 90.000,C 0.000} C_DIS
LIN {X -68.693,Y -28.342,Z -53.151,A -90.000,B 90.000,C 0.000} C_DIS
LIN {X -68.504,Y -28.345,Z -53.077,A -90.000,B 90.000,C 0.000} C_DIS
LIN {X -68.400,Y -28.348,Z -53.039,A -90.000,B 90.000,C 0.000} C_DIS
LIN {X -67.370,Y -28.379,Z -52.696,A -90.000,B 90.000,C 0.000} C_DIS
LIN {X -66.976,Y -28.375,Z -52.541,A -90.000,B 90.000,C 0.000} C_DIS
LIN {X -66.327,Y -28.369,Z -52.291,A -90.000,B 90.000,C 0.000} C_DIS
LIN {X -66.060,Y -28.364,Z -52.176,A -90.000,B 90.000,C 0.000} C_DIS
LIN {X -65.813,Y -28.355,Z -52.071,A -90.000,B 90.000,C 0.000} C_DIS
LIN {X -65.623,Y -28.344,Z -51.991,A -90.000,B 90.000,C 0.000} C_DIS
LIN {X -65.246,Y -28.318,Z -51.835,A -90.000,B 90.000,C 0.000} C_DIS
LIN {X -65.037,Y -28.306,Z -51.758,A -90.000,B 90.000,C 0.000} C_DIS
LIN {X -64.533,Y -28.267,Z -51.591,A -90.000,B 90.000,C 0.000} C_DIS
LIN {X -64.080,Y -28.240,Z -51.439,A -90.000,B 90.000,C 0.000} C_DIS
LIN {X -63.322,Y -28.184,Z -51.188,A -90.000,B 90.000,C 0.000} C_DIS
LIN {X -63.138,Y -28.171,Z -51.135,A -90.000,B 90.000,C 0.000} C_DIS
LIN {X -63.047,Y -28.164,Z -51.111,A -90.000,B 90.000,C 0.000} C_DIS
LIN {X -62.855,Y -28.143,Z -51.068,A -90.000,B 90.000,C 0.000} C_DIS
LIN {X -62.622,Y -28.112,Z -51.018,A -90.000,B 90.000,C 0.000} C_DIS
LIN {X -61.771,Y -28.019,Z -50.828,A -90.000,B 90.000,C 0.000} C_DIS
LIN {X -61.317,Y -27.969,Z -50.730,A -90.000,B 90.000,C 0.000} C_DIS
LIN {X -61.108,Y -27.943,Z -50.692,A -90.000,B 90.000,C 0.000} C_DIS
LIN {X -60.865,Y -27.908,Z -50.659,A -90.000,B 90.000,C 0.000} C_DIS
LIN {X -60.480,Y -27.857,Z -50.620,A -90.000,B 90.000,C 0.000} C_DIS
LIN {X -60.255,Y -27.832,Z -50.606,A -90.000,B 90.000,C 0.000} C_DIS
LIN {X -60.016,Y -27.809,Z -50.592,A -90.000,B 90.000,C 0.000} C_DIS
LIN {X -59.811,Y -27.791,Z -50.579,A -90.000,B 90.000,C 0.000} C_DIS
LIN {X -59.442,Y -27.743,Z -50.563,A -90.000,B 90.000,C 0.000} C_DIS
LIN {X -59.164,Y -27.717,Z -50.546,A -90.000,B 90.000,C 0.000} C_DIS
LIN {X -58.766,Y -27.666,Z -50.530,A -90.000,B 90.000,C 0.000} C_DIS
LIN {X -58.611,Y -27.650,Z -50.528,A -90.000,B 90.000,C 0.000} C_DIS
LIN {X -58.286,Y -27.619,Z -50.529,A -90.000,B 90.000,C 0.000} C_DIS
LIN {X -57.741,Y -27.567,Z -50.531,A -90.000,B 90.000,C 0.000} C_DIS
LIN {X -57.350,Y -27.516,Z -50.540,A -90.000,B 90.000,C 0.000} C_DIS
LIN {X -56.991,Y -27.476,Z -50.563,A -90.000,B 90.000,C 0.000} C_DIS
LIN {X -56.400,Y -27.414,Z -50.607,A -90.000,B 90.000,C 0.000} C_DIS
LIN {X -55.380,Y -27.325,Z -50.674,A -90.000,B 90.000,C 0.000} C_DIS
LIN {X -55.268,Y -27.317,Z -50.684,A -90.000,B 90.000,C 0.000} C_DIS
LIN {X -55.183,Y -27.308,Z -50.693,A -90.000,B 90.000,C 0.000} C_DIS
LIN {X -55.183,Y -60.000,Z -50.693,A -90.000,B 90.000,C 0.000} C_DIS
LIN {X -75.443,Y -60.000,Z -51.216,A -90.000,B 90.000,C 0.000} C_DIS
LIN {X -75.443,Y -27.308,Z -51.216,A -90.000,B 90.000,C 0.000} C_DIS
LIN {X -75.133,Y -27.368,Z -51.410,A -90.000,B 90.000,C 0.000} C_DIS
LIN {X -74.997,Y -27.394,Z -51.501,A -90.000,B 90.000,C 0.000} C_DIS
LIN {X -74.627,Y -27.458,Z -51.733,A -90.000,B 90.000,C 0.000} C_DIS
LIN {X -74.009,Y -27.564,Z -52.111,A -90.000,B 90.000,C 0.000} C_DIS
LIN {X -73.739,Y -27.626,Z -52.279,A -90.000,B 90.000,C 0.000} C_DIS
LIN {X -73.599,Y -27.643,Z -52.286,A -90.000,B 90.000,C 0.000} C_DIS
LIN {X -73.484,Y -27.653,Z -52.267,A -90.000,B 90.000,C 0.000} C_DIS
LIN {X -72.881,Y -27.719,Z -52.164,A -90.000,B 90.000,C 0.000} C_DIS
LIN {X -72.154,Y -27.774,Z -52.055,A -90.000,B 90.000,C 0.000} C_DIS
LIN {X -72.005,Y -27.783,Z -52.019,A -90.000,B 90.000,C 0.000} C_DIS
LIN {X -71.689,Y -27.811,Z -51.941,A -90.000,B 90.000,C 0.000} C_DIS
LIN {X -71.248,Y -27.833,Z -51.846,A -90.000,B 90.000,C 0.000} C_DIS
LIN {X -70.853,Y -27.857,Z -51.762,A -90.000,B 90.000,C 0.000} C_DIS
LIN {X -70.247,Y -27.890,Z -51.605,A -90.000,B 90.000,C 0.000} C_DIS
LIN {X -69.765,Y -27.909,Z -51.445,A -90.000,B 90.000,C 0.000} C_DIS
LIN {X -69.349,Y -27.920,Z -51.309,A -90.000,B 90.000,C 0.000} C_DIS
LIN {X -69.127,Y -27.923,Z -51.223,A -90.000,B 90.000,C 0.000} C_DIS
LIN {X -69.076,Y -27.924,Z -51.205,A -90.000,B 90.000,C 0.000} C_DIS
LIN {X -68.512,Y -27.926,Z -51.019,A -90.000,B 90.000,C 0.000} C_DIS
LIN {X -68.030,Y -27.919,Z -50.863,A -90.000,B 90.000,C 0.000} C_DIS
LIN {X -67.333,Y -27.900,Z -50.596,A -90.000,B 90.000,C 0.000} C_DIS
LIN {X -67.065,Y -27.889,Z -50.495,A -90.000,B 90.000,C 0.000} C_DIS
LIN {X -66.557,Y -27.861,Z -50.281,A -90.000,B 90.000,C 0.000} C_DIS
LIN {X -66.063,Y -27.802,Z -50.083,A -90.000,B 90.000,C 0.000} C_DIS
LIN {X -65.912,Y -27.781,Z -50.027,A -90.000,B 90.000,C 0.000} C_DIS
LIN {X -65.679,Y -27.750,Z -49.947,A -90.000,B 90.000,C 0.000} C_DIS
LIN {X -65.340,Y -27.708,Z -49.840,A -90.000,B 90.000,C 0.000} C_DIS
LIN {X -65.025,Y -27.679,Z -49.737,A -90.000,B 90.000,C 0.000} C_DIS
LIN {X -64.832,Y -27.650,Z -49.678,A -90.000,B 90.000,C 0.000} C_DIS
LIN {X -64.716,Y -27.632,Z -49.642,A -90.000,B 90.000,C 0.000} C_DIS
LIN {X -63.959,Y -27.528,Z -49.409,A -90.000,B 90.000,C 0.000} C_DIS
LIN {X -63.797,Y -27.508,Z -49.364,A -90.000,B 90.000,C 0.000} C_DIS
LIN {X -63.588,Y -27.473,Z -49.314,A -90.000,B 90.000,C 0.000} C_DIS
LIN {X -63.255,Y -27.423,Z -49.243,A -90.000,B 90.000,C 0.000} C_DIS
LIN {X -62.651,Y -27.308,Z -49.128,A -90.000,B 90.000,C 0.000} C_DIS
LIN {X -62.651,Y -60.000,Z -49.128,A -90.000,B 90.000,C 0.000} C_DIS
LIN {X -75.483,Y -60.000,Z -49.216,A -90.000,B 90.000,C 0.000} C_DIS
LIN {X -75.483,Y -27.308,Z -49.216,A -90.000,B 90.000,C 0.000} C_DIS
LIN {X -75.376,Y -27.318,Z -49.217,A -90.000,B 90.000,C 0.000} C_DIS
LIN {X -75.056,Y -27.344,Z -49.254,A -90.000,B 90.000,C 0.000} C_DIS
LIN {X -74.938,Y -27.352,Z -49.281,A -90.000,B 90.000,C 0.000} C_DIS
LIN {X -74.860,Y -27.358,Z -49.303,A -90.000,B 90.000,C 0.000} C_DIS
LIN {X -74.564,Y -27.381,Z -49.421,A -90.000,B 90.000,C 0.000} C_DIS
LIN {X -74.493,Y -27.387,Z -49.458,A -90.000,B 90.000,C 0.000} C_DIS
LIN {X -74.394,Y -27.395,Z -49.515,A -90.000,B 90.000,C 0.000} C_DIS
LIN {X -74.032,Y -27.425,Z -49.742,A -90.000,B 90.000,C 0.000} C_DIS
LIN {X -73.893,Y -27.439,Z -49.833,A -90.000,B 90.000,C 0.000} C_DIS
LIN {X -73.506,Y -27.477,Z -50.074,A -90.000,B 90.000,C 0.000} C_DIS
LIN {X -73.277,Y -27.497,Z -50.214,A -90.000,B 90.000,C 0.000} C_DIS
LIN {X -73.160,Y -27.503,Z -50.196,A -90.000,B 90.000,C 0.000} C_DIS
LIN {X -72.651,Y -27.527,Z -50.121,A -90.000,B 90.000,C 0.000} C_DIS
LIN {X -72.521,Y -27.538,Z -50.101,A -90.000,B 90.000,C 0.000} C_DIS
LIN {X -72.178,Y -27.561,Z -50.017,A -90.000,B 90.000,C 0.000} C_DIS
LIN {X -71.933,Y -27.568,Z -49.964,A -90.000,B 90.000,C 0.000} C_DIS
LIN {X -71.380,Y -27.577,Z -49.848,A -90.000,B 90.000,C 0.000} C_DIS
LIN {X -71.294,Y -27.578,Z -49.831,A -90.000,B 90.000,C 0.000} C_DIS
LIN {X -70.798,Y -27.579,Z -49.707,A -90.000,B 90.000,C 0.000} C_DIS
LIN {X -70.260,Y -27.575,Z -49.533,A -90.000,B 90.000,C 0.000} C_DIS
LIN {X -70.014,Y -27.577,Z -49.454,A -90.000,B 90.000,C 0.000} C_DIS
LIN {X -69.860,Y -27.576,Z -49.395,A -90.000,B 90.000,C 0.000} C_DIS
LIN {X -69.691,Y -27.572,Z -49.335,A -90.000,B 90.000,C 0.000} C_DIS
LIN {X -69.347,Y -27.560,Z -49.224,A -90.000,B 90.000,C 0.000} C_DIS
LIN {X -69.035,Y -27.538,Z -49.126,A -90.000,B 90.000,C 0.000} C_DIS
LIN {X -68.691,Y -27.524,Z -49.017,A -90.000,B 90.000,C 0.000} C_DIS
LIN {X -68.342,Y -27.498,Z -48.887,A -90.000,B 90.000,C 0.000} C_DIS
LIN {X -68.196,Y -27.488,Z -48.832,A -90.000,B 90.000,C 0.000} C_DIS
LIN {X -67.806,Y -27.434,Z -48.693,A -90.000,B 90.000,C 0.000} C_DIS
LIN {X -67.492,Y -27.388,Z -48.569,A -90.000,B 90.000,C 0.000} C_DIS
LIN {X -67.232,Y -27.361,Z -48.463,A -90.000,B 90.000,C 0.000} C_DIS
LIN {X -66.883,Y -27.308,Z -48.326,A -90.000,B 90.000,C 0.000} C_DIS
LIN {X -66.527,Y -27.253,Z -48.181,A -90.000,B 90.000,C 0.000} C_DIS
LIN {X -66.367,Y -27.226,Z -48.112,A -90.000,B 90.000,C 0.000} C_DIS
LIN {X -66.082,Y -27.176,Z -47.979,A -90.000,B 90.000,C 0.000} C_DIS
LIN {X -65.843,Y -27.128,Z -47.854,A -90.000,B 90.000,C 0.000} C_DIS
LIN {X -65.740,Y -27.105,Z -47.794,A -90.000,B 90.000,C 0.000} C_DIS
LIN {X -65.605,Y -27.072,Z -47.708,A -90.000,B 90.000,C 0.000} C_DIS
LIN {X -65.529,Y -27.051,Z -47.653,A -90.000,B 90.000,C 0.000} C_DIS
LIN {X -65.433,Y -27.021,Z -47.574,A -90.000,B 90.000,C 0.000} C_DIS
LIN {X -65.382,Y -27.002,Z -47.523,A -90.000,B 90.000,C 0.000} C_DIS
LIN {X -65.324,Y -26.974,Z -47.451,A -90.000,B 90.000,C 0.000} C_DIS
LIN {X -65.297,Y -26.957,Z -47.405,A -90.000,B 90.000,C 0.000} C_DIS
LIN {X -65.288,Y -26.948,Z -47.382,A -90.000,B 90.000,C 0.000} C_DIS
LIN {X -65.275,Y -26.931,Z -47.339,A -90.000,B 90.000,C 0.000} C_DIS
LIN {X -65.272,Y -26.923,Z -47.317,A -90.000,B 90.000,C 0.000} C_DIS
LIN {X -65.272,Y -26.908,Z -47.276,A -90.000,B 90.000,C 0.000} C_DIS
LIN {X -65.276,Y -26.900,Z -47.256,A -90.000,B 90.000,C 0.000} C_DIS
LIN {X -65.290,Y -26.886,Z -47.218,A -90.000,B 90.000,C 0.000} C_DIS
LIN {X -65.326,Y -26.865,Z -47.162,A -90.000,B 90.000,C 0.000} C_DIS
LIN {X -65.361,Y -26.852,Z -47.128,A -90.000,B 90.000,C 0.000} C_DIS
LIN {X -65.403,Y -26.839,Z -47.094,A -90.000,B 90.000,C 0.000} C_DIS
LIN {X -65.453,Y -26.828,Z -47.062,A -90.000,B 90.000,C 0.000} C_DIS
LIN {X -65.511,Y -26.816,Z -47.032,A -90.000,B 90.000,C 0.000} C_DIS
LIN {X -65.576,Y -26.806,Z -47.003,A -90.000,B 90.000,C 0.000} C_DIS
LIN {X -65.612,Y -26.803,Z -46.989,A -90.000,B 90.000,C 0.000} C_DIS
LIN {X -65.771,Y -26.804,Z -46.937,A -90.000,B 90.000,C 0.000} C_DIS
LIN {X -65.956,Y -26.808,Z -46.891,A -90.000,B 90.000,C 0.000} C_DIS
LIN {X -66.167,Y -26.816,Z -46.849,A -90.000,B 90.000,C 0.000} C_DIS
LIN {X -66.402,Y -26.828,Z -46.813,A -90.000,B 90.000,C 0.000} C_DIS
LIN {X -66.659,Y -26.843,Z -46.782,A -90.000,B 90.000,C 0.000} C_DIS
LIN {X -66.936,Y -26.862,Z -46.755,A -90.000,B 90.000,C 0.000} C_DIS
LIN {X -67.387,Y -26.910,Z -46.723,A -90.000,B 90.000,C 0.000} C_DIS
LIN {X -67.709,Y -26.940,Z -46.707,A -90.000,B 90.000,C 0.000} C_DIS
LIN {X -68.046,Y -26.966,Z -46.695,A -90.000,B 90.000,C 0.000} C_DIS
LIN {X -68.397,Y -26.993,Z -46.687,A -90.000,B 90.000,C 0.000} C_DIS
LIN {X -68.760,Y -27.022,Z -46.683,A -90.000,B 90.000,C 0.000} C_DIS
LIN {X -69.133,Y -27.055,Z -46.682,A -90.000,B 90.000,C 0.000} C_DIS
LIN {X -69.515,Y -27.084,Z -46.684,A -90.000,B 90.000,C 0.000} C_DIS
LIN {X -70.299,Y -27.140,Z -46.697,A -90.000,B 90.000,C 0.000} C_DIS
LIN {X -71.101,Y -27.191,Z -46.720,A -90.000,B 90.000,C 0.000} C_DIS
LIN {X -71.504,Y -27.210,Z -46.735,A -90.000,B 90.000,C 0.000} C_DIS
LIN {X -71.906,Y -27.229,Z -46.753,A -90.000,B 90.000,C 0.000} C_DIS
LIN {X -72.703,Y -27.271,Z -46.792,A -90.000,B 90.000,C 0.000} C_DIS
LIN {X -73.095,Y -27.285,Z -46.815,A -90.000,B 90.000,C 0.000} C_DIS
LIN {X -74.223,Y -27.311,Z -46.888,A -90.000,B 90.000,C 0.000} C_DIS
LIN {X -74.578,Y -27.315,Z -46.913,A -90.000,B 90.000,C 0.000} C_DIS
LIN {X -75.249,Y -27.305,Z -46.966,A -90.000,B 90.000,C 0.000} C_DIS
LIN {X -75.854,Y -27.292,Z -47.020,A -90.000,B 90.000,C 0.000} C_DIS
LIN {X -76.129,Y -27.279,Z -47.046,A -90.000,B 90.000,C 0.000} C_DIS
LIN {X -76.615,Y -27.243,Z -47.097,A -90.000,B 90.000,C 0.000} C_DIS
LIN {X -77.005,Y -27.213,Z -47.144,A -90.000,B 90.000,C 0.000} C_DIS
LIN {X -77.160,Y -27.200,Z -47.165,A -90.000,B 90.000,C 0.000} C_DIS
LIN {X -77.339,Y -27.184,Z -47.195,A -90.000,B 90.000,C 0.000} C_DIS
LIN {X -77.420,Y -27.177,Z -47.212,A -90.000,B 90.000,C 0.000} C_DIS
LIN {X -77.468,Y -27.173,Z -47.228,A -90.000,B 90.000,C 0.000} C_DIS
LIN {X -77.479,Y -27.172,Z -47.235,A -90.000,B 90.000,C 0.000} C_DIS
LIN {X -77.482,Y -27.171,Z -47.241,A -90.000,B 90.000,C 0.000} C_DIS
LIN {X -77.476,Y -27.172,Z -47.247,A -90.000,B 90.000,C 0.000} C_DIS
LIN {X -77.461,Y -27.173,Z -47.252,A -90.000,B 90.000,C 0.000} C_DIS
LIN {X -77.436,Y -27.180,Z -47.257,A -90.000,B 90.000,C 0.000} C_DIS
LIN {X -77.359,Y -27.199,Z -47.264,A -90.000,B 90.000,C 0.000} C_DIS
LIN {X -77.305,Y -27.208,Z -47.266,A -90.000,B 90.000,C 0.000} C_DIS
LIN {X -77.083,Y -27.234,Z -47.269,A -90.000,B 90.000,C 0.000} C_DIS
LIN {X -76.882,Y -27.250,Z -47.267,A -90.000,B 90.000,C 0.000} C_DIS
LIN {X -76.637,Y -27.266,Z -47.261,A -90.000,B 90.000,C 0.000} C_DIS
LIN {X -76.346,Y -27.281,Z -47.252,A -90.000,B 90.000,C 0.000} C_DIS
LIN {X -75.620,Y -27.308,Z -47.221,A -90.000,B 90.000,C 0.000} C_DIS
LIN {X -75.533,Y -27.311,Z -47.217,A -90.000,B 90.000,C 0.000} C_DIS
LIN {X -75.329,Y -27.317,Z -47.218,A -90.000,B 90.000,C 0.000} C_DIS
LIN {X -75.147,Y -27.323,Z -47.230,A -90.000,B 90.000,C 0.000} C_DIS
LIN {X -74.825,Y -27.335,Z -47.268,A -90.000,B 90.000,C 0.000} C_DIS
LIN {X -74.737,Y -27.338,Z -47.280,A -90.000,B 90.000,C 0.000} C_DIS
LIN {X -74.607,Y -27.344,Z -47.305,A -90.000,B 90.000,C 0.000} C_DIS
LIN {X -74.441,Y -27.351,Z -47.344,A -90.000,B 90.000,C 0.000} C_DIS
LIN {X -74.331,Y -27.353,Z -47.375,A -90.000,B 90.000,C 0.000} C_DIS
LIN {X -74.168,Y -27.357,Z -47.427,A -90.000,B 90.000,C 0.000} C_DIS
LIN {X -73.878,Y -27.364,Z -47.542,A -90.000,B 90.000,C 0.000} C_DIS
LIN {X -73.750,Y -27.367,Z -47.594,A -90.000,B 90.000,C 0.000} C_DIS
LIN {X -73.614,Y -27.370,Z -47.661,A -90.000,B 90.000,C 0.000} C_DIS
LIN {X -73.486,Y -27.373,Z -47.730,A -90.000,B 90.000,C 0.000} C_DIS
LIN {X -73.336,Y -27.377,Z -47.818,A -90.000,B 90.000,C 0.000} C_DIS
LIN {X -73.109,Y -27.392,Z -47.960,A -90.000,B 90.000,C 0.000} C_DIS
LIN {X -72.903,Y -27.397,Z -48.091,A -90.000,B 90.000,C 0.000} C_DIS
LIN {X -72.847,Y -27.399,Z -48.128,A -90.000,B 90.000,C 0.000} C_DIS
LIN {X -72.557,Y -27.392,Z -48.060,A -90.000,B 90.000,C 0.000} C_DIS
LIN {X -72.084,Y -27.380,Z -47.962,A -90.000,B 90.000,C 0.000} C_DIS
LIN {X -71.735,Y -27.369,Z -47.891,A -90.000,B 90.000,C 0.000} C_DIS
LIN {X -71.346,Y -27.357,Z -47.795,A -90.000,B 90.000,C 0.000} C_DIS
LIN {X -71.105,Y -27.344,Z -47.719,A -90.000,B 90.000,C 0.000} C_DIS
LIN {X -70.746,Y -27.308,Z -47.607,A -90.000,B 90.000,C 0.000} C_DIS
LIN {X -70.746,Y -60.000,Z -47.607,A -90.000,B 90.000,C 0.000} C_DIS
LIN {X -88.099,Y -60.000,Z -59.800,A -90.000,B 90.000,C 0.000} C_DIS
LIN {X -88.099,Y -27.308,Z -59.800,A -90.000,B 90.000,C 0.000} C_DIS
LIN {X -88.310,Y -27.380,Z -59.517,A -90.000,B 90.000,C 0.000} C_DIS
LIN {X -88.367,Y -27.402,Z -59.436,A -90.000,B 90.000,C 0.000} C_DIS
LIN {X -88.524,Y -27.455,Z -59.200,A -90.000,B 90.000,C 0.000} C_DIS
LIN {X -88.970,Y -27.627,Z -58.493,A -90.000,B 90.000,C 0.000} C_DIS
LIN {X -89.103,Y -27.680,Z -58.264,A -90.000,B 90.000,C 0.000} C_DIS
LIN {X -89.212,Y -27.725,Z -58.072,A -90.000,B 90.000,C 0.000} C_DIS
LIN {X -89.395,Y -27.794,Z -57.730,A -90.000,B 90.000,C 0.000} C_DIS
LIN {X -89.476,Y -27.827,Z -57.573,A -90.000,B 90.000,C 0.000} C_DIS
LIN {X -89.556,Y -27.867,Z -57.402,A -90.000,B 90.000,C 0.000} C_DIS
LIN {X -89.636,Y -27.910,Z -57.225,A -90.000,B 90.000,C 0.000} C_DIS
LIN {X -89.712,Y -27.950,Z -57.033,A -90.000,B 90.000,C 0.000} C_DIS
LIN {X -89.797,Y -28.000,Z -56.797,A -90.000,B 90.000,C 0.000} C_DIS
LIN {X -89.931,Y -28.075,Z -56.412,A -90.000,B 90.000,C 0.000} C_DIS
LIN {X -89.971,Y -28.102,Z -56.284,A -90.000,B 90.000,C 0.000} C_DIS
LIN {X -90.029,Y -28.150,Z -56.071,A -90.000,B 90.000,C 0.000} C_DIS
LIN {X -90.062,Y -28.181,Z -55.905,A -90.000,B 90.000,C 0.000} C_DIS
LIN {X -90.094,Y -28.212,Z -55.725,A -90.000,B 90.000,C 0.000} C_DIS
LIN {X -90.118,Y -28.239,Z -55.569,A -90.000,B 90.000,C 0.000} C_DIS
LIN {X -90.141,Y -28.273,Z -55.389,A -90.000,B 90.000,C 0.000} C_DIS
LIN {X -90.149,Y -28.289,Z -55.307,A -90.000,B 90.000,C 0.000} C_DIS
LIN {X -90.182,Y -28.328,Z -55.088,A -90.000,B 90.000,C 0.000} C_DIS
LIN {X -90.197,Y -28.348,Z -54.942,A -90.000,B 90.000,C 0.000} C_DIS
LIN {X -90.206,Y -28.365,Z -54.817,A -90.000,B 90.000,C 0.000} C_DIS
LIN {X -90.210,Y -28.382,Z -54.684,A -90.000,B 90.000,C 0.000} C_DIS
LIN {X -90.210,Y -28.402,Z -54.545,A -90.000,B 90.000,C 0.000} C_DIS
LIN {X -90.197,Y -28.461,Z -54.077,A -90.000,B 90.000,C 0.000} C_DIS
LIN {X -90.187,Y -28.476,Z -53.937,A -90.000,B 90.000,C 0.000} C_DIS
LIN {X -90.151,Y -28.515,Z -53.559,A -90.000,B 90.000,C 0.000} C_DIS
LIN {X -90.118,Y -28.528,Z -53.354,A -90.000,B 90.000,C 0.000} C_DIS
LIN {X -90.089,Y -28.539,Z -53.198,A -90.000,B 90.000,C 0.000} C_DIS
LIN {X -90.044,Y -28.554,Z -52.989,A -90.000,B 90.000,C 0.000} C_DIS
LIN {X -89.996,Y -28.560,Z -52.810,A -90.000,B 90.000,C 0.000} C_DIS
LIN {X -89.953,Y -28.565,Z -52.670,A -90.000,B 90.000,C 0.000} C_DIS
LIN {X -89.913,Y -28.570,Z -52.553,A -90.000,B 90.000,C 0.000} C_DIS
LIN {X -89.857,Y -28.577,Z -52.412,A -90.000,B 90.000,C 0.000} C_DIS
LIN {X -89.813,Y -28.580,Z -52.306,A -90.000,B 90.000,C 0.000} C_DIS
LIN {X -89.745,Y -28.584,Z -52.155,A -90.000,B 90.000,C 0.000} C_DIS
LIN {X -89.627,Y -28.585,Z -51.916,A -90.000,B 90.000,C 0.000} C_DIS
LIN {X -89.539,Y -28.587,Z -51.755,A -90.000,B 90.000,C 0.000} C_DIS
LIN {X -89.461,Y -28.588,Z -51.618,A -90.000,B 90.000,C 0.000} C_DIS
LIN {X -89.359,Y -28.582,Z -51.458,A -90.000,B 90.000,C 0.000} C_DIS
LIN {X -89.241,Y -28.577,Z -51.293,A -90.000,B 90.000,C 0.000} C_DIS
LIN {X -89.143,Y -28.573,Z -51.167,A -90.000,B 90.000,C 0.000} C_DIS
LIN {X -89.029,Y -28.565,Z -51.034,A -90.000,B 90.000,C 0.000} C_DIS
LIN {X -88.937,Y -28.555,Z -50.936,A -90.000,B 90.000,C 0.000} C_DIS
LIN {X -88.789,Y -28.537,Z -50.789,A -90.000,B 90.000,C 0.000} C_DIS
LIN {X -88.699,Y -28.521,Z -50.703,A -90.000,B 90.000,C 0.000} C_DIS
LIN {X -88.535,Y -28.495,Z -50.561,A -90.000,B 90.000,C 0.000} C_DIS
LIN {X -88.431,Y -28.477,Z -50.475,A -90.000,B 90.000,C 0.000} C_DIS
LIN {X -88.339,Y -28.462,Z -50.407,A -90.000,B 90.000,C 0.000} C_DIS
LIN {X -88.229,Y -28.445,Z -50.331,A -90.000,B 90.000,C 0.000} C_DIS
LIN {X -88.134,Y -28.429,Z -50.270,A -90.000,B 90.000,C 0.000} C_DIS
LIN {X -88.058,Y -28.417,Z -50.224,A -90.000,B 90.000,C 0.000} C_DIS
LIN {X -87.915,Y -28.382,Z -50.146,A -90.000,B 90.000,C 0.000} C_DIS
LIN {X -87.785,Y -28.351,Z -50.082,A -90.000,B 90.000,C 0.000} C_DIS
LIN {X -87.371,Y -28.253,Z -49.881,A -90.000,B 90.000,C 0.000} C_DIS
LIN {X -87.181,Y -28.209,Z -49.794,A -90.000,B 90.000,C 0.000} C_DIS
LIN {X -87.079,Y -28.184,Z -49.750,A -90.000,B 90.000,C 0.000} C_DIS
LIN {X -86.713,Y -28.073,Z -49.616,A -90.000,B 90.000,C 0.000} C_DIS
LIN {X -86.516,Y -28.017,Z -49.555,A -90.000,B 90.000,C 0.000} C_DIS
LIN {X -86.469,Y -28.002,Z -49.543,A -90.000,B 90.000,C 0.000} C_DIS
LIN {X -86.359,Y -27.965,Z -49.518,A -90.000,B 90.000,C 0.000} C_DIS
LIN {X -86.223,Y -27.922,Z -49.492,A -90.000,B 90.000,C 0.000} C_DIS
LIN {X -85.987,Y -27.853,Z -49.458,A -90.000,B 90.000,C 0.000} C_DIS
LIN {X -85.659,Y -27.756,Z -49.427,A -90.000,B 90.000,C 0.000} C_DIS
LIN {X -85.437,Y -27.690,Z -49.420,A -90.000,B 90.000,C 0.000} C_DIS
LIN {X -85.269,Y -27.645,Z -49.423,A -90.000,B 90.000,C 0.000} C_DIS
LIN {X -85.162,Y -27.617,Z -49.428,A -90.000,B 90.000,C 0.000} C_DIS
LIN {X -84.982,Y -27.569,Z -49.445,A -90.000,B 90.000,C 0.000} C_DIS
LIN {X -84.732,Y -27.507,Z -49.474,A -90.000,B 90.000,C 0.000} C_DIS
LIN {X -84.598,Y -27.475,Z -49.492,A -90.000,B 90.000,C 0.000} C_DIS
LIN {X -84.447,Y -27.443,Z -49.517,A -90.000,B 90.000,C 0.000} C_DIS
LIN {X -84.350,Y -27.424,Z -49.535,A -90.000,B 90.000,C 0.000} C_DIS
LIN {X -84.272,Y -27.404,Z -49.553,A -90.000,B 90.000,C 0.000} C_DIS
LIN {X -84.130,Y -27.372,Z -49.589,A -90.000,B 90.000,C 0.000} C_DIS
LIN {X -83.815,Y -27.308,Z -49.676,A -90.000,B 90.000,C 0.000} C_DIS
LIN {X -83.815,Y -60.000,Z -49.676,A -90.000,B 90.000,C 0.000} C_DIS
LIN {X -91.847,Y -60.000,Z -56.136,A -90.000,B 90.000,C 0.000} C_DIS
LIN {X -91.847,Y -27.308,Z -56.136,A -90.000,B 90.000,C 0.000} C_DIS
LIN {X -91.926,Y -27.413,Z -55.811,A -90.000,B 90.000,C 0.000} C_DIS
LIN {X -91.957,Y -27.460,Z -55.668,A -90.000,B 90.000,C 0.000} C_DIS
LIN {X -92.000,Y -27.535,Z -55.399,A -90.000,B 90.000,C 0.000} C_DIS
LIN {X -92.024,Y -27.569,Z -55.263,A -90.000,B 90.000,C 0.000} C_DIS
LIN {X -92.057,Y -27.621,Z -55.061,A -90.000,B 90.000,C 0.000} C_DIS
LIN {X -92.080,Y -27.669,Z -54.882,A -90.000,B 90.000,C 0.000} C_DIS
LIN {X -92.095,Y -27.712,Z -54.728,A -90.000,B 90.000,C 0.000} C_DIS
LIN {X -92.098,Y -27.722,Z -54.687,A -90.000,B 90.000,C 0.000} C_DIS
LIN {X -92.106,Y -27.777,Z -54.429,A -90.000,B 90.000,C 0.000} C_DIS
LIN {X -92.107,Y -27.831,Z -54.182,A -90.000,B 90.000,C 0.000} C_DIS
LIN {X -92.103,Y -27.898,Z -53.853,A -90.000,B 90.000,C 0.000} C_DIS
LIN {X -92.095,Y -27.935,Z -53.675,A -90.000,B 90.000,C 0.000} C_DIS
LIN {X -92.084,Y -27.957,Z -53.537,A -90.000,B 90.000,C 0.000} C_DIS
LIN {X -92.066,Y -27.988,Z -53.322,A -90.000,B 90.000,C 0.000} C_DIS
LIN {X -92.054,Y -28.001,Z -53.221,A -90.000,B 90.000,C 0.000} C_DIS
LIN {X -92.016,Y -28.035,Z -52.960,A -90.000,B 90.000,C 0.000} C_DIS
LIN {X -91.981,Y -28.061,Z -52.761,A -90.000,B 90.000,C 0.000} C_DIS
LIN {X -91.934,Y -28.084,Z -52.536,A -90.000,B 90.000,C 0.000} C_DIS
LIN {X -91.911,Y -28.098,Z -52.434,A -90.000,B 90.000,C 0.000} C_DIS
LIN {X -91.864,Y -28.117,Z -52.248,A -90.000,B 90.000,C 0.000} C_DIS
LIN {X -91.796,Y -28.128,Z -52.027,A -90.000,B 90.000,C 0.000} C_DIS
LIN {X -91.754,Y -28.141,Z -51.900,A -90.000,B 90.000,C 0.000} C_DIS
LIN {X -91.681,Y -28.155,Z -51.706,A -90.000,B 90.000,C 0.000} C_DIS
LIN {X -91.591,Y -28.160,Z -51.493,A -90.000,B 90.000,C 0.000} C_DIS
LIN {X -91.565,Y -28.160,Z -51.434,A -90.000,B 90.000,C 0.000} C_DIS
LIN {X -91.511,Y -28.166,Z -51.314,A -90.000,B 90.000,C 0.000} C_DIS
LIN {X -91.437,Y -28.172,Z -51.162,A -90.000,B 90.000,C 0.000} C_DIS
LIN {X -91.329,Y -28.171,Z -50.951,A -90.000,B 90.000,C 0.000} C_DIS
LIN {X -91.279,Y -28.166,Z -50.862,A -90.000,B 90.000,C 0.000} C_DIS
LIN {X -91.203,Y -28.168,Z -50.726,A -90.000,B 90.000,C 0.000} C_DIS
LIN {X -91.145,Y -28.168,Z -50.625,A -90.000,B 90.000,C 0.000} C_DIS
LIN {X -91.015,Y -28.162,Z -50.419,A -90.000,B 90.000,C 0.000} C_DIS
LIN {X -90.963,Y -28.159,Z -50.342,A -90.000,B 90.000,C 0.000} C_DIS
LIN {X -90.903,Y -28.157,Z -50.256,A -90.000,B 90.000,C 0.000} C_DIS
LIN {X -90.786,Y -28.143,Z -50.099,A -90.000,B 90.000,C 0.000} C_DIS
LIN {X -90.659,Y -28.130,Z -49.940,A -90.000,B 90.000,C 0.000} C_DIS
LIN {X -90.526,Y -28.107,Z -49.788,A -90.000,B 90.000,C 0.000} C_DIS
LIN {X -90.366,Y -28.080,Z -49.620,A -90.000,B 90.000,C 0.000} C_DIS
LIN {X -90.112,Y -28.036,Z -49.373,A -90.000,B 90.000,C 0.000} C_DIS
LIN {X -90.012,Y -28.017,Z -49.281,A -90.000,B 90.000,C 0.000} C_DIS
LIN {X -89.913,Y -27.999,Z -49.196,A -90.000,B 90.000,C 0.000} C_DIS
LIN {X -89.767,Y -27.960,Z -49.078,A -90.000,B 90.000,C 0.000} C_DIS
LIN {X -89.629,Y -27.920,Z -48.974,A -90.000,B 90.000,C 0.000} C_DIS
LIN {X -89.482,Y -27.881,Z -48.873,A -90.000,B 90.000,C 0.000} C_DIS
LIN {X -89.369,Y -27.850,Z -48.798,A -90.000,B 90.000,C 0.000} C_DIS
LIN {X -89.182,Y -27.799,Z -48.687,A -90.000,B 90.000,C 0.000} C_DIS
LIN {X -89.024,Y -27.759,Z -48.600,A -90.000,B 90.000,C 0.000} C_DIS
LIN {X -88.868,Y -27.711,Z -48.521,A -90.000,B 90.000,C 0.000} C_DIS
LIN {X -88.643,Y -27.643,Z -48.417,A -90.000,B 90.000,C 0.000} C_DIS
LIN {X -88.455,Y -27.579,Z -48.334,A -90.000,B 90.000,C 0.000} C_DIS
LIN {X -88.340,Y -27.536,Z -48.284,A -90.000,B 90.000,C 0.000} C_DIS
LIN {X -88.284,Y -27.513,Z -48.262,A -90.000,B 90.000,C 0.000} C_DIS
LIN {X -87.978,Y -27.383,Z -48.153,A -90.000,B 90.000,C 0.000} C_DIS
LIN {X -87.841,Y -27.325,Z -48.110,A -90.000,B 90.000,C 0.000} C_DIS
LIN {X -87.801,Y -27.308,Z -48.098,A -90.000,B 90.000,C 0.000} C_DIS
LIN {X -87.638,Y -27.244,Z -48.051,A -90.000,B 90.000,C 0.000} C_DIS
LIN {X -87.407,Y -27.151,Z -47.992,A -90.000,B 90.000,C 0.000} C_DIS
LIN {X -87.263,Y -27.094,Z -47.960,A -90.000,B 90.000,C 0.000} C_DIS
LIN {X -87.060,Y -27.012,Z -47.924,A -90.000,B 90.000,C 0.000} C_DIS
LIN {X -86.872,Y -26.937,Z -47.901,A -90.000,B 90.000,C 0.000} C_DIS
LIN {X -86.701,Y -26.870,Z -47.890,A -90.000,B 90.000,C 0.000} C_DIS
LIN {X -86.545,Y -26.814,Z -47.891,A -90.000,B 90.000,C 0.000} C_DIS
LIN {X -86.449,Y -26.784,Z -47.898,A -90.000,B 90.000,C 0.000} C_DIS
LIN {X -86.318,Y -26.751,Z -47.919,A -90.000,B 90.000,C 0.000} C_DIS
LIN {X -86.238,Y -26.738,Z -47.939,A -90.000,B 90.000,C 0.000} C_DIS
LIN {X -86.165,Y -26.731,Z -47.964,A -90.000,B 90.000,C 0.000} C_DIS
LIN {X -86.131,Y -26.731,Z -47.978,A -90.000,B 90.000,C 0.000} C_DIS
LIN {X -86.067,Y -26.735,Z -48.010,A -90.000,B 90.000,C 0.000} C_DIS
LIN {X -86.010,Y -26.747,Z -48.046,A -90.000,B 90.000,C 0.000} C_DIS
LIN {X -85.983,Y -26.755,Z -48.066,A -90.000,B 90.000,C 0.000} C_DIS
LIN {X -85.934,Y -26.777,Z -48.109,A -90.000,B 90.000,C 0.000} C_DIS
LIN {X -85.891,Y -26.806,Z -48.156,A -90.000,B 90.000,C 0.000} C_DIS
LIN {X -85.872,Y -26.822,Z -48.181,A -90.000,B 90.000,C 0.000} C_DIS
LIN {X -85.838,Y -26.860,Z -48.235,A -90.000,B 90.000,C 0.000} C_DIS
LIN {X -85.809,Y -26.904,Z -48.292,A -90.000,B 90.000,C 0.000} C_DIS
LIN {X -85.786,Y -26.953,Z -48.353,A -90.000,B 90.000,C 0.000} C_DIS
LIN {X -85.768,Y -27.007,Z -48.418,A -90.000,B 90.000,C 0.000} C_DIS
LIN {X -85.755,Y -27.065,Z -48.487,A -90.000,B 90.000,C 0.000} C_DIS
LIN {X -85.748,Y -27.127,Z -48.559,A -90.000,B 90.000,C 0.000} C_DIS
LIN {X -85.745,Y -27.191,Z -48.634,A -90.000,B 90.000,C 0.000} C_DIS
LIN {X -85.748,Y -27.258,Z -48.713,A -90.000,B 90.000,C 0.000} C_DIS
LIN {X -85.755,Y -27.327,Z -48.795,A -90.000,B 90.000,C 0.000} C_DIS
LIN {X -85.775,Y -27.433,Z -48.923,A -90.000,B 90.000,C 0.000} C_DIS
LIN {X -85.795,Y -27.504,Z -49.013,A -90.000,B 90.000,C 0.000} C_DIS
LIN {X -85.847,Y -27.647,Z -49.200,A -90.000,B 90.000,C 0.000} C_DIS
LIN {X -85.916,Y -27.799,Z -49.396,A -90.000,B 90.000,C 0.000} C_DIS
LIN {X -86.002,Y -27.959,Z -49.602,A -90.000,B 90.000,C 0.000} C_DIS
LIN {X -86.050,Y -28.037,Z -49.709,A -90.000,B 90.000,C 0.000} C_DIS
LIN {X -86.103,Y -28.112,Z -49.817,A -90.000,B 90.000,C 0.000} C_DIS
LIN {X -86.160,Y -28.184,Z -49.927,A -90.000,B 90.000,C 0.000} C_DIS
LIN {X -86.220,Y -28.252,Z -50.038,A -90.000,B 90.000,C 0.000} C_DIS
LIN {X -86.283,Y -28.316,Z -50.152,A -90.000,B 90.000,C 0.000} C_DIS
LIN {X -86.350,Y -28.377,Z -50.266,A -90.000,B 90.000,C 0.000} C_DIS
LIN {X -86.420,Y -28.434,Z -50.383,A -90.000,B 90.000,C 0.000} C_DIS
LIN {X -86.494,Y -28.488,Z -50.500,A -90.000,B 90.000,C 0.000} C_DIS
LIN {X -86.650,Y -28.594,Z -50.738,A -90.000,B 90.000,C 0.000} C_DIS
LIN {X -86.733,Y -28.647,Z -50.859,A -90.000,B 90.000,C 0.000} C_DIS
LIN {X -86.818,Y -28.695,Z -50.980,A -90.000,B 90.000,C 0.000} C_DIS
LIN {X -86.906,Y -28.737,Z -51.102,A -90.000,B 90.000,C 0.000} C_DIS
LIN {X -86.997,Y -28.775,Z -51.224,A -90.000,B 90.000,C 0.000} C_DIS
LIN {X -87.091,Y -28.807,Z -51.347,A -90.000,B 90.000,C 0.000} C_DIS
LIN {X -87.186,Y -28.834,Z -51.471,A -90.000,B 90.000,C 0.000} C_DIS
LIN {X -87.284,Y -28.855,Z -51.594,A -90.000,B 90.000,C 0.000} C_DIS
LIN {X -87.592,Y -28.902,Z -51.965,A -90.000,B 90.000,C 0.000} C_DIS
LIN {X -87.698,Y -28.913,Z -52.089,A -90.000,B 90.000,C 0.000} C_DIS
LIN {X -87.806,Y -28.918,Z -52.212,A -90.000,B 90.000,C 0.000} C_DIS
LIN {X -87.916,Y -28.918,Z -52.334,A -90.000,B 90.000,C 0.000} C_DIS
LIN {X -88.028,Y -28.914,Z -52.456,A -90.000,B 90.000,C 0.000} C_DIS
LIN {X -88.141,Y -28.904,Z -52.577,A -90.000,B 90.000,C 0.000} C_DIS
LIN {X -88.371,Y -28.879,Z -52.817,A -90.000,B 90.000,C 0.000} C_DIS
LIN {X -88.725,Y -28.827,Z -53.169,A -90.000,B 90.000,C 0.000} C_DIS
LIN {X -88.846,Y -28.804,Z -53.284,A -90.000,B 90.000,C 0.000} C_DIS
LIN {X -88.967,Y -28.776,Z -53.397,A -90.000,B 90.000,C 0.000} C_DIS
LIN {X -89.088,Y -28.754,Z -53.509,A -90.000,B 90.000,C 0.000} C_DIS
LIN {X -89.211,Y -28.727,Z -53.618,A -90.000,B 90.000,C 0.000} C_DIS
LIN {X -89.580,Y -28.629,Z -53.936,A -90.000,B 90.000,C 0.000} C_DIS
LIN {X -89.704,Y -28.592,Z -54.038,A -90.000,B 90.000,C 0.000} C_DIS
LIN {X -89.952,Y -28.511,Z -54.235,A -90.000,B 90.000,C 0.000} C_DIS
LIN {X -90.076,Y -28.471,Z -54.329,A -90.000,B 90.000,C 0.000} C_DIS
LIN {X -90.199,Y -28.426,Z -54.421,A -90.000,B 90.000,C 0.000} C_DIS
LIN {X -90.446,Y -28.331,Z -54.596,A -90.000,B 90.000,C 0.000} C_DIS
LIN {X -90.568,Y -28.283,Z -54.679,A -90.000,B 90.000,C 0.000} C_DIS
LIN {X -90.690,Y -28.231,Z -54.759,A -90.000,B 90.000,C 0.000} C_DIS
LIN {X -90.812,Y -28.175,Z -54.836,A -90.000,B 90.000,C 0.000} C_DIS
LIN {X -91.052,Y -28.054,Z -54.980,A -90.000,B 90.000,C 0.000} C_DIS
LIN {X -91.288,Y -27.935,Z -55.109,A -90.000,B 90.000,C 0.000} C_DIS
LIN {X -91.405,Y -27.874,Z -55.168,A -90.000,B 90.000,C 0.000} C_DIS
LIN {X -91.520,Y -27.810,Z -55.223,A -90.000,B 90.000,C 0.000} C_DIS
LIN {X -91.633,Y -27.746,Z -55.274,A -90.000,B 90.000,C 0.000} C_DIS
LIN {X -91.856,Y -27.616,Z -55.364,A -90.000,B 90.000,C 0.000} C_DIS
LIN {X -91.965,Y -27.553,Z -55.402,A -90.000,B 90.000,C 0.000} C_DIS
LIN {X -92.178,Y -27.433,Z -55.465,A -90.000,B 90.000,C 0.000} C_DIS
LIN {X -92.332,Y -27.346,Z -55.500,A -90.000,B 90.000,C 0.000} C_DIS
LIN {X -92.432,Y -27.289,Z -55.517,A -90.000,B 90.000,C 0.000} C_DIS
LIN {X -92.530,Y -27.235,Z -55.529,A -90.000,B 90.000,C 0.000} C_DIS
LIN {X -92.626,Y -27.182,Z -55.536,A -90.000,B 90.000,C 0.000} C_DIS
LIN {X -92.765,Y -27.108,Z -55.536,A -90.000,B 90.000,C 0.000} C_DIS
LIN {X -92.854,Y -27.062,Z -55.530,A -90.000,B 90.000,C 0.000} C_DIS
LIN {X -92.941,Y -27.021,Z -55.518,A -90.000,B 90.000,C 0.000} C_DIS
LIN {X -93.025,Y -26.983,Z -55.501,A -90.000,B 90.000,C 0.000} C_DIS
LIN {X -93.106,Y -26.949,Z -55.477,A -90.000,B 90.000,C 0.000} C_DIS
LIN {X -93.184,Y -26.921,Z -55.448,A -90.000,B 90.000,C 0.000} C_DIS
LIN {X -93.259,Y -26.897,Z -55.413,A -90.000,B 90.000,C 0.000} C_DIS
LIN {X -93.331,Y -26.878,Z -55.372,A -90.000,B 90.000,C 0.000} C_DIS
LIN {X -93.400,Y -26.864,Z -55.324,A -90.000,B 90.000,C 0.000} C_DIS
LIN {X -93.465,Y -26.855,Z -55.271,A -90.000,B 90.000,C 0.000} C_DIS
LIN {X -93.526,Y -26.851,Z -55.210,A -90.000,B 90.000,C 0.000} C_DIS
LIN {X -93.584,Y -26.853,Z -55.144,A -90.000,B 90.000,C 0.000} C_DIS
LIN {X -93.639,Y -26.860,Z -55.070,A -90.000,B 90.000,C 0.000} C_DIS
LIN {X -93.690,Y -26.872,Z -54.990,A -90.000,B 90.000,C 0.000} C_DIS
LIN {X -93.736,Y -26.889,Z -54.903,A -90.000,B 90.000,C 0.000} C_DIS
LIN {X -93.779,Y -26.908,Z -54.808,A -90.000,B 90.000,C 0.000} C_DIS
LIN {X -93.835,Y -26.942,Z -54.654,A -90.000,B 90.000,C 0.000} C_DIS
LIN {X -93.868,Y -26.970,Z -54.541,A -90.000,B 90.000,C 0.000} C_DIS
LIN {X -93.896,Y -26.999,Z -54.422,A -90.000,B 90.000,C 0.000} C_DIS
LIN {X -93.919,Y -27.033,Z -54.295,A -90.000,B 90.000,C 0.000} C_DIS
LIN {X -93.939,Y -27.075,Z -54.160,A -90.000,B 90.000,C 0.000} C_DIS
LIN {X -93.953,Y -27.117,Z -54.017,A -90.000,B 90.000,C 0.000} C_DIS
LIN {X -93.963,Y -27.159,Z -53.866,A -90.000,B 90.000,C 0.000} C_DIS
LIN {X -93.968,Y -27.201,Z -53.708,A -90.000,B 90.000,C 0.000} C_DIS
LIN {X -93.967,Y -27.244,Z -53.541,A -90.000,B 90.000,C 0.000} C_DIS
LIN {X -93.958,Y -27.308,Z -53.276,A -90.000,B 90.000,C 0.000} C_DIS
LIN {X -93.944,Y -27.368,Z -53.023,A -90.000,B 90.000,C 0.000} C_DIS
LIN {X -93.921,Y -27.410,Z -52.810,A -90.000,B 90.000,C 0.000} C_DIS
LIN {X -93.889,Y -27.460,Z -52.558,A -90.000,B 90.000,C 0.000} C_DIS
LIN {X -93.839,Y -27.515,Z -52.258,A -90.000,B 90.000,C 0.000} C_DIS
LIN {X -93.797,Y -27.556,Z -52.034,A -90.000,B 90.000,C 0.000} C_DIS
LIN {X -93.722,Y -27.593,Z -51.724,A -90.000,B 90.000,C 0.000} C_DIS
LIN {X -93.646,Y -27.628,Z -51.455,A -90.000,B 90.000,C 0.000} C_DIS
LIN {X -93.586,Y -27.646,Z -51.270,A -90.000,B 90.000,C 0.000} C_DIS
LIN {X -93.557,Y -27.654,Z -51.185,A -90.000,B 90.000,C 0.000} C_DIS
LIN {X -93.487,Y -27.669,Z -50.997,A -90.000,B 90.000,C 0.000} C_DIS
LIN {X -93.421,Y -27.682,Z -50.833,A -90.000,B 90.000,C 0.000} C_DIS
LIN {X -93.349,Y -27.697,Z -50.659,A -90.000,B 90.000,C 0.000} C_DIS
LIN {X -93.259,Y -27.705,Z -50.459,A -90.000,B 90.000,C 0.000} C_DIS
LIN {X -93.211,Y -27.705,Z -50.362,A -90.000,B 90.000,C 0.000} C_DIS
LIN {X -93.096,Y -27.715,Z -50.130,A -90.000,B 90.000,C 0.000} C_DIS
LIN {X -92.985,Y -27.714,Z -49.921,A -90.000,B 90.000,C 0.000} C_DIS
LIN {X -92.932,Y -27.708,Z -49.829,A -90.000,B 90.000,C 0.000} C_DIS
LIN {X -92.794,Y -27.705,Z -49.592,A -90.000,B 90.000,C 0.000} C_DIS
LIN {X -92.665,Y -27.695,Z -49.390,A -90.000,B 90.000,C 0.000} C_DIS
LIN {X -92.593,Y -27.684,Z -49.284,A -90.000,B 90.000,C 0.000} C_DIS
LIN {X -92.440,Y -27.672,Z -49.070,A -90.000,B 90.000,C 0.000} C_DIS
LIN {X -92.373,Y -27.664,Z -48.980,A -90.000,B 90.000,C 0.000} C_DIS
LIN {X -92.284,Y -27.653,Z -48.866,A -90.000,B 90.000,C 0.000} C_DIS
LIN {X -92.199,Y -27.643,Z -48.760,A -90.000,B 90.000,C 0.000} C_DIS
LIN {X -92.020,Y -27.610,Z -48.555,A -90.000,B 90.000,C 0.000} C_DIS
LIN {X -91.925,Y -27.589,Z -48.454,A -90.000,B 90.000,C 0.000} C_DIS
LIN {X -91.815,Y -27.564,Z -48.341,A -90.000,B 90.000,C 0.000} C_DIS
LIN {X -91.580,Y -27.513,Z -48.114,A -90.000,B 90.000,C 0.000} C_DIS
LIN {X -91.427,Y -27.465,Z -47.977,A -90.000,B 90.000,C 0.000} C_DIS
LIN {X -91.320,Y -27.430,Z -47.886,A -90.000,B 90.000,C 0.000} C_DIS
LIN {X -91.117,Y -27.367,Z -47.724,A -90.000,B 90.000,C 0.000} C_DIS
LIN {X -90.954,Y -27.308,Z -47.604,A -90.000,B 90.000,C 0.000} C_DIS
LIN {X -90.954,Y -60.000,Z -47.604,A -90.000,B 90.000,C 0.000} C_DIS
LIN {X -74.270,Y -60.000,Z -73.481,A -90.000,B 90.000,C 0.000} C_DIS
LIN {X -74.270,Y -27.308,Z -73.481,A -90.000,B 90.000,C 0.000} C_DIS
LIN {X -74.586,Y -27.348,Z -73.201,A -90.000,B 90.000,C 0.000} C_DIS
LIN {X -74.770,Y -27.361,Z -73.052,A -90.000,B 90.000,C 0.000} C_DIS
LIN {X -74.785,Y -27.364,Z -73.041,A -90.000,B 90.000,C 0.000} C_DIS
LIN {X -74.827,Y -27.376,Z -73.015,A -90.000,B 90.000,C 0.000} C_DIS
LIN {X -74.991,Y -27.417,Z -72.926,A -90.000,B 90.000,C 0.000} C_DIS
LIN {X -75.165,Y -27.472,Z -72.839,A -90.000,B 90.000,C 0.000} C_DIS
LIN {X -75.424,Y -27.431,Z -72.899,A -90.000,B 90.000,C 0.000} C_DIS
LIN {X -75.595,Y -27.402,Z -72.935,A -90.000,B 90.000,C 0.000} C_DIS
LIN {X -75.828,Y -27.371,Z -72.980,A -90.000,B 90.000,C 0.000} C_DIS
LIN {X -76.133,Y -27.334,Z -73.031,A -90.000,B 90.000,C 0.000} C_DIS
LIN {X -76.358,Y -27.308,Z -73.064,A -90.000,B 90.000,C 0.000} C_DIS
LIN {X -76.358,Y -60.000,Z -73.064,A -90.000,B 90.000,C 0.000} C_DIS
LIN {X -1.626,Y -60.000,Z -168.076,A -90.000,B 90.000,C 0.000} C_DIS
LIN {X -1.626,Y -60.000,Z -168.076,A -90.000,B 90.000,C 0.000} C_DIS
LIN {X -1.627,Y -27.308,Z -168.076,A -90.000,B 90.000,C 0.000} C_DIS
LIN {X -1.559,Y -27.328,Z -167.881,A -90.000,B 90.000,C 0.000} C_DIS
LIN {X -1.369,Y -27.349,Z -167.056,A -90.000,B 90.000,C 0.000} C_DIS
LIN {X -1.294,Y -27.340,Z -166.596,A -90.000,B 90.000,C 0.000} C_DIS
LIN {X -1.116,Y -27.339,Z -165.457,A -90.000,B 90.000,C 0.000} C_DIS
LIN {X -1.118,Y -27.326,Z -165.324,A -90.000,B 90.000,C 0.000} C_DIS
LIN {X -1.158,Y -27.324,Z -164.769,A -90.000,B 90.000,C 0.000} C_DIS
LIN {X -1.208,Y -27.325,Z -164.094,A -90.000,B 90.000,C 0.000} C_DIS
LIN {X -1.240,Y -27.308,Z -164.016,A -90.000,B 90.000,C 0.000} C_DIS
LIN {X -1.240,Y -60.000,Z -164.016,A -90.000,B 90.000,C 0.000} C_DIS
LIN {X -103.702,Y -60.000,Z -243.561,A -90.000,B 90.000,C 0.000} C_DIS
LIN {X -103.702,Y -27.308,Z -243.561,A -90.000,B 90.000,C 0.000} C_DIS
LIN {X -101.457,Y -27.308,Z -241.944,A -90.000,B 90.000,C 0.000} C_DIS
LIN {X -98.714,Y -27.308,Z -240.105,A -90.000,B 90.000,C 0.000} C_DIS
LIN {X -93.789,Y -27.308,Z -236.722,A -90.000,B 90.000,C 0.000} C_DIS
LIN {X -93.242,Y -27.308,Z -236.364,A -90.000,B 90.000,C 0.000} C_DIS
LIN {X -91.524,Y -27.308,Z -235.255,A -90.000,B 90.000,C 0.000} C_DIS
